	11:
		TON_Abblasdauer(IN := TRUE, PT := Abblasdauer);

		IF 	TON_Abblasdauer.Q
			AND Q_DWORD = 0
		THEN
			state 											:= 10;
		ELSE
			IF 	NOT TOF_Abblastakt.Q 
				AND Q_DWORD <> 0 
			THEN
				TOF_Abblastakt(IN:=TRUE  , PT:= Abblastakt);
				Q_DWORD 									:= 0;
			ELSIF	NOT TOF_Abblastakt.Q 
					AND Q_DWORD = 0 
			THEN
				TOF_Abblastakt(IN:= TRUE , PT:= Abblastakt) ;
				Q_DWORD 									:= SETBIT32(Q_DWORD,i);
			END_IF
			(* Work Timer *)
			TOF_Abblastakt(IN:=FALSE);
		END_IF

	END_CASE
ELSE
	Aktiv 													:= FALSE;
	state 													:= 0;
	Q_DWORD													:= 0;
END_IF

(**********************************************************************************************************)

END_FUNCTION_BLOCK

// ---- POUs/Axis_PTPV3_CoE.TcPOU
FUNCTION_BLOCK Axis_PTPV3_CoE
VAR_OUTPUT CONSTANT
	MIN_JOB													:	INT := 0;
	MAX_JOB													:	INT := 5;
END_VAR
VAR_INPUT
(* Ax Move cmd Parameter *)
	JobId													:	INT := MIN_JOB;
	Job														:	ARRAY[MIN_JOB..MAX_JOB] OF AX_JOB;

(* Axis *)
	ref														:	AXIS_REF; (* siehe Lib TcMc2 *)
	Admin													: 	Ax_AdminCtrl ; (* PTP Ax Control Baustein *)
	para													: 	Ax_Para; (* Achsparameter lesen/schreiben *)
	Motion													:	Ax_MotionCtrl;
	Home													:	Ax_HomingCtrl;
	HMI														:	Ax_HMI;
	Gear				:	Ax_GearCtrl;
	rMasterAxis											:	REFERENCE TO AXIS_REF := 0;
	
(* Ax Optionsmodule *)
	(* Drive *)
	drive													:	Ax_CanOpenDriveEventCtrl;

	(* Error Handling *)
	errorNC													:	Ax_ErrorNCEventCtrl;
                                                    	
	AutoFctCtrl												:	Ax_AutoFctCtrl; (* Softwareendlagen und Refernzierflag ein/ausschalten *)
END_VAR                                             	
VAR_OUTPUT                                          	
	ErrHdl													:	ERROR_HDL;
	EventStatus												:	BYTE;
//	HmiStatus												:	BYTE;
//	startName												:	STRING(10);
//	statusTxt												:	STRING(MAX_STRING_LENGTH);
END_VAR
VAR
	i 														: 	INT;
END_VAR

	(* Axis 																*)
	(************************************************************************)

(* work IO **********************************************************************)


(********************************************************************************)
(* work Admin ctrl 																*)
(********************************************************************************)
	Admin(
		RST			:= , 
		Enable		:= ,
		EnablePos	:= ,
		EnableNeg	:= ,
		BufferMode:= ,
		Override	:= ,
		rAxis		:= Ref,
		ShowNCErrIfDisabled := ,
		EnableOK	=> ,
		Ready		=> ,
		StartRel	=> ,
		Busy		=> ,
		Done		=> ,
		Error		=> ,
		ErrorID		=> );
		
(********************************************************************************)
(* work homing ctrl 															*)
(********************************************************************************)
	Home(
		Execute		:= ,
		Fnc			:= ,
		BufferMode	:= ,
		Mode		:= ,
		AcceptBlockedDrive:= ,
		CalibrationCam:= ,
		Pos			:= ,
		SetPosModeRel:= ,
		SetPosOptions:= ,
		rAxis		:= Ref,
		FNC_HOMING	=> ,
		FNC_HALT	=> ,
		FNC_SETPOS	=> ,
		Active		=> ,
		Done		=> ,
		Busy		=> ,
		CmdAborted	=> ,
		Error		=> ,
		ErrorId		=> ,
		ErrorText	=> );

(********************************************************************************)
(* work moving ctrl 															*)
(********************************************************************************)
	Motion(
		Execute		:= ,
		Fnc			:= ,
		JogFwd		:= ,
		JogBwd		:= ,
		BufferMode	:= ,
		Direction	:= ,
		JogMode		:= ,
		Target		:= ,
		Velo		:= ,
		Jerk		:= ,
		Acc			:= ,
		Dec			:= ,
		MoveOptions:= ,
		rAxis		:= Ref,
		FNC_STOP	=> ,
		FNC_HALT	=> ,
		FNC_MOVE_JOG	=> ,
		FNC_MOVE_ABS	=> ,
		FNC_MOVE_REL	=> ,
		FNC_MOVE_ADD	=> ,
		FNC_MOVE_MOD	=> ,
		FNC_MOVE_VELO	=> ,
		Active		=> ,
		Done		=> ,
		Busy		=> ,
		CmdAborted	=> ,
		Error		=> ,
		ErrorId		=> ,
		ErrorText	=> );

(********************************************************************************)
(* Achse Koppeln 																*)
(********************************************************************************)
(*
	Gear(
		Execute		:= ,
		Fnc			:= ,
		RatioDyn	:= ,
		RatioNumerator:= ,
		RatioDenominator:= ,
		Acc			:= ,
		pMasterAxis1:= ,
		pMasterAxis2:= ,
		pMasterAxis3:= ,
		pMasterAxis4:= ,
		MasterGearRatio1:= ,
		MasterGearRatio2:= ,
		MasterGearRatio3:= ,
		MasterGearRatio4:= ,
		rAxis		:= REF,
		FNC_GEAR_OUT=> ,
		FNC_GEAR_IN=> ,
		FNC_GEAR_IN_DYN=> ,
		FNC_GEAR_IN_MM=> ,
		InGear		=> ,
		Active		=> ,
		Done		=> ,
		Busy		=> ,
		CmdAborted=> ,
		Error		=> ,
		ErrorId		=> ,
		ErrorText	=> );
*)
(********************************************************************************)
(* Parameter																	*)
(*******************************************************************************
	para(
		Execute		:= ,
		Fnc			:= ,
		AxID		:= ref.NcToPlc.AxisId,
		InitDone	=> ,
		Done		=> ,
		Busy		=> ,
		Error		=> );
*)

(******************************************************************************)
(* Hilfsfunktionen der Achse(Setzen,Rücksetzen von Ref.flag und Softwareendl.)*)
(******************************************************************************)
	AutoFctCtrl(
		enable				:= NOT AutoFctCtrl.Error AND Para.InitDone,
		axId				:= ref.NcToPlc.AxisId,
		forceSoftLimit		:= ref.Status.Homed OR para.EncTypAbs = 1, (* nicht referenziert oder Encodertyp Abs. *)
		forceCalibration	:= , //Siehe Abblikation 
		Status				=> ,
		Busy				=> ,
		Error				=> ,
		ErrorId				=> );

(********************************************************************************)
(* Error NC																		*)
(********************************************************************************)
	IF Admin.Error
	THEN
		ErrHdl.id 		:= UDINT_TO_DINT(Admin.ErrorId);
		ErrHdl.fnc		:= 'Admin';
		ErrHdl.text		:= Admin.ErrorText;
		ErrHdl.flag		:= TRUE;
	ELSIF Motion.Error
	THEN
		ErrHdl.id 		:= UDINT_TO_DINT(Motion.ErrorId);
		ErrHdl.fnc		:= 'Motion';
		ErrHdl.text		:= Motion.ErrorText;
		ErrHdl.flag		:= TRUE;
	ELSIF Home.Error
	THEN
		ErrHdl.id 		:= UDINT_TO_DINT(Home.ErrorId);
		ErrHdl.fnc		:= 'Home';
		ErrHdl.text		:= Home.ErrorText;
		ErrHdl.flag		:= TRUE;

(*	ELSIF Gear.Error
	THEN
		ErrHdl.id 		:= UDINT_TO_DINT(gear.ErrorId);
		ErrHdl.fnc		:= 'Gear';
		ErrHdl.text		:= Gear.ErrorText;
		ErrHdl.flag		:= TRUE;
*)
	ELSE
		ErrHdl.Reset();
	END_IF
	
	errorNC(
		Enable			:=	Admin.EnableOK,
		InAck			:= NOT Errhdl.flag AND errorNC.StatusByte <> 0 OR Admin.RST,
		Name			:= para.Name,
		SourceId		:= (* Default *) ,
		rAxis			:= ref,
		AxErrorId		:= DINT_TO_UDINT(ErrHdl.Id),
		CmdAborted		:= ,
		StatusByte		=> ,
		SOURCE_AXIS		=> );
		
(********************************************************************************)
(* Drive 																		*)
(********************************************************************************)
	drive(
		EnableEvent		:= , 
		InAck			:= errorNC.InAck, 
		Name			:= para.Name, 
		ErrorEndlagePos:= , 
		ErrorEndlageNeg:= , 
		ErrorSchutzschalter:= , 
		rAxis			:= ref, 
		Busy			=> , 
		Error			=> , 
		ErrorId			=> , 
		Fault			=> , 
		Ready			=> , 
		LiveCountTimeout=> , 
		LiveCount		=> , 
		RT_StatusChanged=> , 
		CanNodeSTATE	=> , 
		EventStatusByte	=> , 
		SOURCE_DRIVES_CAN=> );
		
(* Event Status *****************************************************************)
	EventStatus																:= 	errorNC.StatusByte
																				OR Drive.EventStatusByte;
		
(* Check start arr pos **********************************************************)
	CheckTargetPos();

(********************************************************************************)
(* Hmi Axis				 														*)
(********************************************************************************)
	HMI(Motion := Motion);
	
	Gear(
	FNC_GEAR_OUT=> , 
	FNC_GEAR_IN=> , 
	FNC_GEAR_IN_DYN=> , 
	FNC_GEAR_IN_MM=> , 
	Execute:= , 
	Fnc:= , 
	RatioDyn:= , 
	RatioNumerator:= , 
	RatioDenominator:= , 
	Acc:= , 
	Options:= , 
	rMasterAxis1:=rMasterAxis , 		//直接写
	rMasterAxis2:= , 
	rMasterAxis3:= , 
	rMasterAxis4:= , 
	MasterGearRatio1:= , 
	MasterGearRatio2:= , 
	MasterGearRatio3:= , 
	MasterGearRatio4:= , 
	rAxis:= ref, 
	Active=> , 
	Done=> , 
	Busy=> , 
	CmdAborted=> , 
	Error=> , 
	ErrorId=> , 
	ErrorText=> );
	
	
(*
	HmiStatus.0 := ref.Status.NegativeDirection;
	HmiStatus.1 := ref.Status.PositiveDirection;
	HmiStatus.2 := ref.Status.InTargetPosition  ;
	HmiStatus.3 := ref.Status.Homed;
	HmiStatus.4 := Admin.EnableNeg; 
	HmiStatus.5 := Admin.EnablePos;
	HmiStatus.6 := Admin.Ready;
	HmiStatus.7 := ErrHdl.flag;
*)
(* Set Status Txt ***************************************************************)
(*	IF Pulse._1s.RT THEN
		statusTxt := CONCAT(para.Name,' Id:');
		statusTxt := CONCAT(statusTxt,DWORD_TO_STRING(ref.NcToPlc.AxisId));
		statusTxt := CONCAT(statusTxt,SEL(ctrl.Ready,',NOT Ready,Istpos:',',Ready,Istpos:'));
		statusTxt := CONCAT(statusTxt,LREAL_TO_FMTSTR(ctrl.ActPos, 2, TRUE));
		statusTxt := CONCAT(statusTxt,',Target:');
		statusTxt := CONCAT(statusTxt,LREAL_TO_FMTSTR(ctrl.Target, 2, TRUE));
		(* Zeilenwechsel *)
		statusTxt := CONCAT(statusTxt,'$r');
		(* ------------- *)
		statusTxt := CONCAT(statusTxt,SEL(ctrl.NotMoving,SEL(ref.Status.PositiveDirection,',Moving NEG,StartId:',',Moving POS,StartId:'),',NOT Moving,StartId:'));
		statusTxt := CONCAT(statusTxt,INT_TO_STRING(StartID));
		statusTxt := CONCAT(statusTxt,',ErrorId:');
		statusTxt := CONCAT(statusTxt,DINT_TO_STRING(ctrl.ErrHdl.id));
		statusTxt := CONCAT(statusTxt,',Cmd:');
		statusTxt := CONCAT(statusTxt,INT_TO_STRING(ctrl.Cmd));
		statusTxt := CONCAT(statusTxt,',ActCmd:');
		statusTxt := CONCAT(statusTxt,INT_TO_STRING(ctrl.Actcmd));
	END_IF
*)


(***********************************************************************************************)

METHOD PUBLIC CheckTargetPos
VAR_INPUT
END_VAR
FOR i := MIN_JOB TO MAX_JOB DO
	IF Job[i].Fnc = 6 THEN
		Job[i].InTarget := REF.Status.NotMoving
									AND(
									REF.NcToPlc.ModuloActPos >= Job[i].Target - para.Zielfenster
									AND REF.NcToPlc.ModuloActPos <= Job[i].Target + para.Zielfenster
									OR
									(MODABS(Job[i].Target,para.ModuloFaktor) <= 0 + para.Zielfenster
									OR MODABS(Job[i].Target,para.ModuloFaktor) >= para.ModuloFaktor - para.Zielfenster)
									AND(
									REF.NcToPlc.ModuloActPos >= para.ModuloFaktor - para.Zielfenster
									OR REF.NcToPlc.ModuloActPos <= 0 + para.Zielfenster));

		Job[i].InPosWindow	:= REF.NcToPlc.ModuloActPos >= Job[i].Target - para.Posfenster
									AND REF.NcToPlc.ModuloActPos <= Job[i].Target + para.Posfenster
									OR
									(MODABS(Job[i].Target,para.ModuloFaktor) <= 0 + para.Posfenster
									OR MODABS(Job[i].Target,para.ModuloFaktor) >= para.ModuloFaktor - para.Posfenster)
									AND(
									REF.NcToPlc.ModuloActPos >= para.ModuloFaktor - para.Posfenster
									OR REF.NcToPlc.ModuloActPos <= 0 + para.Posfenster);
	ELSE
		Job[i].InTarget := REF.Status.NotMoving
									AND REF.NcToPlc.ActPos >= Job[i].Target - para.Zielfenster
									AND REF.NcToPlc.ActPos <= Job[i].Target + para.Zielfenster ;

		Job[i].InPosWindow	:= REF.NcToPlc.ActPos >= Job[i].Target - para.Posfenster
									AND REF.NcToPlc.ActPos <= Job[i].Target + para.Posfenster;
	END_IF
END_FOR
END_METHOD

METHOD PUBLIC NoAction : BOOL //Result = Busy of home , gear , motion , ....
VAR_INPUT
END_VAR
home.Execute	:= FALSE;
//gear.Execute	:= FALSE;
Motion.Execute	:= FALSE;
Motion.JogBwd	:= FALSE;
Motion.JogFwd	:= FALSE;
Gear.Execute	:=FALSE;

NoAction 		:= NOT home.Busy
					AND NOT gear.Busy
					and not Motion.Busy;
END_METHOD

METHOD PUBLIC reset
VAR_INPUT
END_VAR
Admin.Reset(FALSE);
drive.Ack();
errorNC.Ack();
END_METHOD

METHOD PUBLIC StartMotion
VAR_INPUT
	JobID			:	int ;
END_VAR
THIS^.JobID		:= Jobid;

IF JobID >= MIN_JOB AND JobId <= MAX_JOB
THEN
	CheckTargetPos();
//	startName				:= Job[Jobid].name;
	Motion.Fnc 				:= Job[Jobid].Fnc;
	Motion.BufferMode 		:= Job[Jobid].BufferMode;
	Motion.Direction 		:= Job[Jobid].Direction;
	Motion.Target 			:= Job[Jobid].Target;
	Motion.Velo 			:= Job[Jobid].Velo;
	Admin.Override 			:= Job[Jobid].Override;
	Motion.Acc		 		:= Job[Jobid].Acc;
	Motion.Dec				:= Job[Jobid].Dec;
	Motion.Jerk	 			:= Job[Jobid].Jerk;
	MOtion.Execute			:= TRUE;
END_IF
END_METHOD

END_FUNCTION_BLOCK

// ---- POUs/PTP/01_Base/Ax_MotionCtrl.TcPOU
{attribute 'no_check'}
FUNCTION_BLOCK Ax_MotionCtrl (* Achse reseten,BTB schalten, starten und stoppen *)
(* A C H T U N G !!!
	For performance reasons the MC-function-blocks MC_MoveRelative, MC_MoveAdditive, MC_MoveVelocity and 
	MC_MoveModulo are commented out insed the declaration.
	If needed, the comment-signs can be removed.

	Alle Bausteine sind schon ausprogrammiert und können in vollem Umfang benutzt werden.
	(MC_MoveAbsolute ->  MC_MoveRelative mit BufferMode-Aborting -> MC_MoveAdditive mit BufferMode-MC_BlendingLow ... 

*)  
VAR_OUTPUT CONSTANT
	FNC_HALT												:	INT := 0;
	FNC_STOP												:	INT := 1;
	FNC_MOVE_JOG											:	INT := 2;
	FNC_MOVE_ABS											:	INT := 3;
	FNC_MOVE_REL											:	INT := 4;
	FNC_MOVE_ADD											:	INT := 5;
	FNC_MOVE_MOD											:	INT := 6;
	FNC_MOVE_VELO											:	INT := 7;
END_VAR
VAR_INPUT
	Execute													:	BOOL := FALSE;
	Fnc														:	INT (FNC_HALT..FNC_MOVE_VELO) := FNC_HALT;
	JogFwd													:	BOOL := FALSE;
	JogBwd													:	BOOL	:= FALSE;
	BufferMode												:	MC_BufferMode := MC_Aborting;(* 	MC_Aborting,
																											MC_Buffered,
																											MC_BlendingLow,
																											MC_BlendingPrevious,
																											MC_BlendingNext,
																											MC_BlendingHigh *)
	Direction												:	MC_Direction := MC_POSITIVE_DIRECTION;	(*	MC_POSITIVE_DIRECTION,
																														   MC_SHORTeSTATE.WAY,
																														   MC_NEGATIVE_DIRECTION,
																														   MC_CURRENT_DIRECTION *)
	JogMode													:	E_JogMode := MC_JOGMODE_STANDARD_SLOW;	(*	MC_JOGMODE_STANDARD_SLOW
																															MC_JOGMODE_STANDARD_FAST
																															MC_JOGMODE_CONTINOUS
																															MC_JOGMODE_INCHING 
																															MC_JOGeMODE.INCHING_MODULO *)
	Target													:	LREAL; (* Zielposition *)
	Velo														: 	LREAL; (* Zielgeschwindigkeit *)
	Jerk														:	LREAL := 0.0; (* Bei 0 werden wird der Ruck aus dem TCManager uebernommen *)
	Acc														:	LREAL := 0.0; (* Bei 0 werden wird die Beschleunigung aus dem TCManager uebernommen *)
	Dec														:	LREAL := 0.0; (* Bei 0 werden wird die Verzoegerung aus dem TCManager uebernommen *)
	MoveOptions												:	ST_MoveOptions;
	rAxis														:	REFERENCE TO AXIS_REF := 0;
END_VAR                     								
VAR_IN_OUT                  								
END_VAR                     								
VAR_OUTPUT                  								
	Active													:	BOOL;
	Done													:	BOOL;
	Busy													:	BOOL;
	CmdAborted												:	BOOL;
	Error													:	BOOL;
	ErrorId													:	UDINT;
	ErrorText												:	STRING(40);
END_VAR
VAR
(* Zwischenspeicher **************************************************************************)
	MemFnc													:	INT := -1;
	MemFncAct												:	INT := -1;
	MCFctTxt												:	STRING(25);
	TrigID													:	INT := 2; (* um mit Trig 1 zu starten *)
	MemBufferMode											:	MC_BufferMode;
	ActSetTarget											:	LREAL;
	ActSetVelo												:	LREAL;
	BusyIntern												:	BOOL;

(* Timer *)

(* Trigger *)
	rtExecute												:	R_TRIG;
	rtExecuteMethod											:	R_TRIG;

(* Instanzierung der MC Bausteine *******************************************************)
	MC_Halt													: 	MC_Halt;
	MC_Stop													: 	MC_Stop;
	MC_MoveVeloPreTrig										: 	MC_MoveVelocity;
	MC_Jog													: 	MC_Jog;

(* Durch entfernen der Kommentarsymbole koennen noch weitere benötigte MC_Move Varianten
	mit ins Programm genommen werden 
*)
	MC_MoveAbsolute											: 	ARRAY[1..2] OF MC_MoveAbsolute;
	MC_MoveModulo											: 	ARRAY[1..2] OF MC_MoveModulo;
	MC_MoveRelative											: 	ARRAY[1..2] OF MC_MoveRelative;
	MC_MoveAdditive											: 	ARRAY[1..2] OF MC_MoveAdditive; 
	MC_MoveVelocity											: 	ARRAY[1..2] OF MC_MoveVelocity; 

(* Dummy Speicher **********************************************************)
	i														: INT := 0 ;

(* Skalierungsfaktor ermitteln *********************************************
	Skalierungsfaktor von 0.1 eintragen. Istpositon "Anfang" merken.
	Antrieb um einen realen Wert "X" mm verfahren. Differenz der
	momentanen Istposition zur Istposition "Anfang" ermitteln.
	SKalierungsfaktor =		realer Fahrweg 
							---------------------------
							Differenz der Istpositionen
*)
END_VAR

	(****************************************************************************************)
	(*																						*)
	(*		B E C K H O F F   N E W   A U T O M A T I O N   T E C H N O L O G Y    			*)
	(*																						*)
	(*		Eiserstr.5	D-33415 Verl	Germany	phone:	+49-5246-0	www.Beckhoff.Com		*)
    (*																						*)
    (*		Bausteinbeschreibung	:	Ax Move Ctrl										*)
	(*		TwinCAT-Version			:	3.x or higher										*)
	(*		Lib						:	TcMC2.lib Newest Version!							*)
	(*		Version					:	V1.2												*)
 	(*		Autor					:	Daniel Schlingmann									*)
	(*																						*)
	(*		Changelog:																		*)
	(*		12.07.14	-	Kein Signal CmdAborted von MC_Jog wenn Software Endl erreicht	*)
	(****************************************************************************************)

(* Execute ***************************************************************************************)
	rtExecute(CLK := Execute XOR(JogBwd AND NOT JogFwd OR JogFwd AND NOT JogBwd));
	
	IF rtExecute.Q
	THEN
		MemFnc 												:= SEL(JogBwd OR JogFwd, Fnc, FNC_MOVE_JOG) ;
		Busy												:= TRUE;
		Done												:= FALSE;
		Active												:= FALSE;
		Error												:= FALSE;
		ErrorID												:= 0;
		CmdAborted											:= FALSE;
		ErrorText											:= '';
	END_IF

(* Call Method ***********************************************************************************)
	CASE MemFnc OF
	FNC_STOP												:	Stop(Execute);
	FNC_HALT												:	Halt(Execute);
	FNC_MOVE_JOG											:	MoveJog(Execute);
	FNC_MOVE_ABS											:	MoveAbs(Execute);
	FNC_MOVE_REL											:	MoveRel(Execute);
	FNC_MOVE_ADD											:	MoveAdd(Execute);
	FNC_MOVE_MOD											:	MoveMod(Execute);
	FNC_MOVE_VELO											:	MoveVelo(Execute);
	-1:
		IF NOT Execute
		THEN
			Busy											:= FALSE;
			Done											:= FALSE;
			Error											:= FALSE;
			ErrorID											:= 0;
			Active											:= FALSE;
			CmdAborted										:= FALSE;
			ErrorText										:= '';
		END_IF
	ELSE
		Busy												:= FALSE;
		Done												:= FALSE;
		Active												:= FALSE;
		Error												:= Execute;
		ErrorID												:= 1803;
		CmdAborted											:= FALSE;
		ErrorText											:= CONCAT('invalid parameter value(s) Fnc no: ' , INT_TO_STRING(MemFnc));
	END_CASE

(*************************************************************************************************)

METHOD PRIVATE _MCIntern
VAR_INPUT
END_VAR
(* Internal MC Action											*)
(****************************************************************)

(* Check Pointer **********************************************************************)
IF NOT __ISVALIDREF(rAxis) 
THEN
	Busy													:= NOT Error;
	Error													:= TRUE;
	ErrorId													:= 16#4B30;
	CmdAborted												:= FALSE;
	Done														:= FALSE;
	Active													:= FALSE;
	ErrorText												:= 'Reference rAxis invalid (0)';
	MemFnc													:= SEL(Execute , -1 ,MemFnc); 
	RETURN;
END_IF

(* flag Execute ***********************************************************************)
	rtExecuteMethod(CLK := Execute OR rtExecute.Q);
	IF rtExecuteMethod.Q
	THEN
		MC_Stop.Execute										:= FALSE;
		MC_Halt.Execute										:=	FALSE;
		MC_MoveVeloPreTrig.Execute							:= FALSE;
		MC_MoveModulo[1].Execute 							:= MC_MoveModulo[2].Execute	:= FALSE;
		MC_MoveAbsolute[1].Execute							:= MC_MoveAbsolute[2].Execute	:= FALSE;
		MC_MoveRelative[1].Execute 							:= MC_MoveRelative[2].Execute := FALSE; 
		MC_MoveAdditive[1].Execute 							:= MC_MoveAdditive[2].Execute := FALSE; 
		MC_MoveVelocity[1].Execute 							:= MC_MoveVelocity[2].Execute := FALSE; 
		BusyIntern											:= FALSE;
		MemFncAct 											:= MemFnc;
	END_IF

(* ctrl programm ******************************************************************************)
	CASE MemFncAct OF
	-1: ; //No Fnc started
	FNC_STOP:
		MC_Stop.Execute										:=	Execute; (* Achse Locked solange Stop noch ansteht *)
		MC_Stop.Deceleration 								:= Dec;
		MC_Stop.Jerk 										:= Jerk;
		MC_Stop.Options 									:= MoveOptions;

	FNC_HALT:
		MC_Halt.Execute										:=	NOT MC_Stop.Busy AND Execute; (* Execute if axis is not locked *)
		MC_Halt.BufferMode									:= BufferMode;
		MC_Halt.Deceleration 								:= Dec;
		MC_Halt.Jerk 										:= Jerk;
		MC_Halt.Options 									:= MoveOptions;
		BusyIntern											:= MC_Stop.Busy;

	FNC_MOVE_JOG:
		IF(Execute OR JogBwd OR JogFwd OR MC_Halt.Busy) (* new cmd or stop last cmd busy *)
			AND NOT rAxis.NcToPlc.StateDWord.2  (* NotMoving *)
			AND NOT MC_Jog.Busy (* not if Mc_Jog running *)
			AND NOT rAxis.NcToPlc.StateDWord.5 (* Protected *) (* not if axis coupled or in NCI group *)
			AND NOT MC_Halt.Error AND NOT MC_Halt.CommandAborted
		THEN
			MC_Halt.Execute									:=	TRUE;
			MC_Halt.BufferMode								:= MC_Aborting;
			MC_Halt.Deceleration 							:= Dec;
			MC_Halt.Jerk 									:= Jerk;
			MC_Halt.Options 								:= MoveOptions;
			BusyIntern										:= TRUE;
		ELSE
			MC_Jog.JogBackwards								:= NOT MC_Stop.Busy AND (JogBwd XOR Execute AND Direction = MC_NEGATIVE_DIRECTION);
			MC_Jog.JogForward								:= NOT MC_Stop.Busy AND (JogFwd XOR Execute AND Direction = MC_POSITIVE_DIRECTION);
			MC_Jog.Mode										:= JogMode;
			MC_Jog.Position 								:= Target;
			MC_Jog.Velocity 								:= Velo;
			MC_Jog.Acceleration 							:= Acc;
			MC_Jog.Deceleration 							:= Dec;
			MC_Jog.Jerk 									:= Jerk;
			MC_Halt.Execute									:=	FALSE;
			BusyIntern										:= MC_Stop.Busy;
		END_IF

	FNC_MOVE_ABS..FNC_MOVE_VELO:
		IF MC_Stop.Busy
			OR rAxis.NcToPlc.StateDWord.29 (* MotionCommandsLocked *)
			OR MC_Jog.Busy
		THEN (* Solange hier rein bis Achse wieder frei und Stop nicht mehr Busy *)
			BusyIntern										:= TRUE;

		ELSIF rAxis.NcToPlc.StateDWord.24 (* CmdBuffered *) 
		THEN (* this section is for aborting a buffered running axis *)
			IF NOT MC_MoveVeloPreTrig.Execute
				AND BufferMode = MC_Aborting
				AND(
				rtExecuteMethod.Q (* new cmd with MC_Aborting zu break up current and buffered cmd *)
				OR 		(* or break up current and buffered cmd with new targetpos. *)
				Execute
				AND (Busy OR Done OR CmdAborted) (* dont restart if error is active *)
				AND (ActSetTarget <> Target))
			THEN
				TrigID 										:= 0;
				MC_MoveVeloPreTrig.Execute 					:= TRUE;
				MC_MoveVeloPreTrig.BufferMode 				:= MC_Aborting;
				MC_MoveVeloPreTrig.Velocity 				:= Velo;
				IF rAxis.NcToPlc.StateDWord.10 (* NegativeDirection *) 
				THEN
					MC_MoveVeloPreTrig.Direction 			:= MC_NEGATIVE_DIRECTION;
				ELSE
					MC_MoveVeloPreTrig.Direction 			:= MC_POSITIVE_DIRECTION;
				END_IF
				BusyIntern									:= TRUE;
			ELSE
				;
			END_IF

		ELSE (* ready for start/restart (MC_MoveVeloPreTrig is active) *)
			IF rtExecuteMethod.Q (* new cmd *)
				OR TrigID = 0 (* new cmd with Buffermode aborted *)
				OR(	Execute
				AND (Busy OR Done OR CmdAborted) (* dont restart if error is active *)
				AND (ActSetTarget <> Target OR ActSetVelo <> Velo AND BufferMode = MC_Aborting)) (* restart only with new velo if bufferMode = Aborting *)
			THEN (* new cmd *)
				(* Cancel MoveVeloPreTrig block *)
				IF TrigID = 0 THEN
					MemBufferMode 							:= MC_Aborting;
				ELSE
					MemBufferMode						 	:= BufferMode;
				END_IF

				(* change TrigID *)
				IF TrigID <> 1 THEN
					TrigID 									:= 1;
				ELSE
					TrigID 									:= 2;
				END_IF

				(* Save Act. target and velo *)
				ActSetTarget 								:= Target;
				ActSetVelo 									:= Velo;

				(* Init MC-Blocks *)
				MC_MoveModulo[1].Execute 					:= MC_MoveModulo[2].Execute	:= FALSE;
				MC_MoveAbsolute[1].Execute					:= MC_MoveAbsolute[2].Execute	:= FALSE;
				MC_MoveRelative[1].Execute 					:= MC_MoveRelative[2].Execute := FALSE; 
				MC_MoveAdditive[1].Execute 					:= MC_MoveAdditive[2].Execute := FALSE; 
				MC_MoveVelocity[1].Execute 					:= MC_MoveVelocity[2].Execute := FALSE; 
			END_IF

			CASE MemFncAct OF
			FNC_MOVE_ABS:(* Absolute *);
				MC_MoveAbsolute[TrigID].Execute				:= Execute OR BusyIntern;
				MC_MoveAbsolute[TrigID].BufferMode 			:= MemBufferMode;
				MC_MoveAbsolute[TrigID].Position 			:= Target;
				MC_MoveAbsolute[TrigID].Velocity 			:= Velo;
				MC_MoveAbsolute[TrigID].Acceleration 		:= Acc;
				MC_MoveAbsolute[TrigID].Deceleration 		:= Dec;
				MC_MoveAbsolute[TrigID].Jerk 				:= Jerk;
				MC_MoveAbsolute[TrigID].Options 			:= MoveOptions;

			FNC_MOVE_MOD:(* Modulo *);
				MC_MoveModulo[TrigID].Execute				:= Execute OR BusyIntern;
				MC_MoveModulo[TrigID].BufferMode 			:= MemBufferMode;
				MC_MoveModulo[TrigID].Position 				:= Target;
				MC_MoveModulo[TrigID].Direction 			:= Direction;
				MC_MoveModulo[TrigID].Velocity 				:= Velo;
				MC_MoveModulo[TrigID].Acceleration 			:= Acc;
				MC_MoveModulo[TrigID].Deceleration 			:= Dec;
				MC_MoveModulo[TrigID].Jerk 					:= Jerk;
				MC_MoveModulo[TrigID].Options 				:= MoveOptions;
			
			FNC_MOVE_REL: (* Relativ *)
				MC_MoveRelative[TrigID].Execute				:= Execute OR BusyIntern;
				MC_MoveRelative[TrigID].BufferMode 			:= MemBufferMode;
				MC_MoveRelative[TrigID].Distance 			:= Target;
				MC_MoveRelative[TrigID].Velocity 			:= Velo;
				MC_MoveRelative[TrigID].Acceleration 		:= Acc;
				MC_MoveRelative[TrigID].Deceleration	 	:= Dec;
				MC_MoveRelative[TrigID].Jerk 				:= Jerk;
				MC_MoveRelative[TrigID].Options 			:= MoveOptions;
		
			FNC_MOVE_ADD:(* Rel.Additive *);
				MC_MoveAdditive[TrigID].Execute				:= Execute OR BusyIntern;
				MC_MoveAdditive[TrigID].BufferMode 			:= MemBufferMode;
				MC_MoveAdditive[TrigID].Distance 			:= Target;
				MC_MoveAdditive[TrigID].Velocity 			:= Velo;
				MC_MoveAdditive[TrigID].Acceleration	 	:= Acc;
				MC_MoveAdditive[TrigID].Deceleration	 	:= Dec;
				MC_MoveAdditive[TrigID].Jerk 				:= Jerk;
				MC_MoveAdditive[TrigID].Options 			:= MoveOptions;
			
			FNC_MOVE_VELO:(* Velocity *);
				MC_MoveVelocity[TrigID].Execute				:= Execute OR BusyIntern;
				MC_MoveVelocity[TrigID].BufferMode 			:= MemBufferMode;
				MC_MoveVelocity[TrigID].Direction 			:= Direction;
				MC_MoveVelocity[TrigID].Velocity 			:= Velo;
				MC_MoveVelocity[TrigID].Acceleration 		:= Acc;
				MC_MoveVelocity[TrigID].Deceleration 		:= Dec;
				MC_MoveVelocity[TrigID].Jerk 				:= Jerk;
				MC_MoveVelocity[TrigID].Options 			:= MoveOptions;
			
			ELSE
				MC_Halt.Execute								:=	TRUE; // axis locked as long as Stop is set 
				Error										:= TRUE;
				ErrorId										:= 16#1803;
				ErrorText									:= CONCAT('invalid parameter value(s) - Fnc no ', INT_TO_STRING(MemFncAct)) ;
			END_CASE

			(* Reset busy intern *)
			MC_MoveVeloPreTrig.Execute 						:= FALSE;
			BusyIntern										:= FALSE;
		END_IF
	ELSE
		MC_Halt.Execute										:=	TRUE; // axis locked as long as Stop is set
		Error												:= TRUE;
		ErrorId												:= 16#1803;
		ErrorText											:= CONCAT('invalid parameter value(s) - Fnc no ', INT_TO_STRING(MemFncAct)) ;
	END_CASE

(****************************************************************************)
(* Work MC Blocks 															*)
(****************************************************************************)

	(* Halt/Stop *)
	MC_Stop(Axis	:= rAxis);
	MC_Halt(Axis	:= rAxis);

	(* Jog *)
	IF MC_Jog.JogBackwards OR MC_Jog.JogForward OR MC_Jog.Busy
		OR MC_Jog.Done OR MC_Jog.Active
		OR MC_Jog.CommandAborted OR MC_Jog.Error
	THEN
		MC_Jog( Axis :=	rAxis);
		MC_Jog.JogBackwards									:= FALSE;
		MC_Jog.JogForward									:= FALSE;
	END_IF

	(* Positionierungen ********************************************)
	(* MC Move Velo PreTrig 1 *)
	IF MC_MoveVeloPreTrig.Execute OR MC_MoveVeloPreTrig.Busy
		OR MC_MoveVeloPreTrig.InVelocity OR MC_MoveVeloPreTrig.Active
		OR MC_MoveVeloPreTrig.CommandAborted OR MC_MoveVeloPreTrig.Error
	THEN
		MC_MoveVeloPreTrig(Axis	:=	rAxis);
	END_IF

	(* Run MC *)
	IF MC_MoveAbsolute[1].Execute OR MC_MoveAbsolute[1].Busy
		OR MC_MoveAbsolute[1].Done OR MC_MoveAbsolute[1].Active
		OR MC_MoveAbsolute[1].CommandAborted OR MC_MoveAbsolute[1].Error
	THEN
		MC_MoveAbsolute[1]( Axis	:=	rAxis);
	END_IF

	IF MC_MoveModulo[1].Execute OR MC_MoveModulo[1].Busy
		OR MC_MoveModulo[1].Done OR MC_MoveModulo[1].Active
		OR MC_MoveModulo[1].CommandAborted OR MC_MoveModulo[1].Error
	THEN
		MC_MoveModulo[1](Axis	:=	rAxis);
	END_IF
	
	IF MC_MoveRelative[1].Execute OR MC_MoveRelative[1].Busy
		OR MC_MoveRelative[1].Done OR MC_MoveRelative[1].Active
		OR MC_MoveRelative[1].CommandAborted OR MC_MoveRelative[1].Error
	THEN
		MC_MoveRelative[1](Axis	:=	rAxis);
	END_IF
	
	IF MC_MoveAdditive[1].Execute OR MC_MoveAdditive[1].Busy
		OR MC_MoveAdditive[1].Done OR MC_MoveAdditive[1].Active
		OR MC_MoveAdditive[1].CommandAborted OR MC_MoveAdditive[1].Error
	THEN
		MC_MoveAdditive[1](Axis	:=	rAxis);
	END_IF
	
	IF MC_MoveVelocity[1].Execute OR MC_MoveVelocity[1].Busy
		OR MC_MoveVelocity[1].Active OR MC_MoveVelocity[1].InVelocity
		OR MC_MoveVelocity[1].CommandAborted OR MC_MoveVelocity[1].Error
	THEN
		MC_MoveVelocity[1](Axis	:=	rAxis);
	END_IF

	(* MC Move Velo PreTrig 2 **************************************)
	(* Run Trig 2 *)
	IF MC_MoveAbsolute[2].Execute OR MC_MoveAbsolute[2].Busy
		OR MC_MoveAbsolute[2].Done OR MC_MoveAbsolute[2].Active
		OR MC_MoveAbsolute[2].CommandAborted OR MC_MoveAbsolute[2].Error
	THEN
		MC_MoveAbsolute[2](Axis	:=	rAxis);
	END_IF

	IF MC_MoveModulo[2].Execute OR MC_MoveModulo[2].Busy
		OR MC_MoveModulo[2].Done OR MC_MoveModulo[2].Active
		OR MC_MoveModulo[2].CommandAborted OR MC_MoveModulo[2].Error
	THEN
		MC_MoveModulo[2](Axis	:=	rAxis);
	END_IF

	
	IF MC_MoveRelative[2].Execute OR MC_MoveRelative[2].Busy
		OR MC_MoveRelative[2].Done OR MC_MoveRelative[2].Active
		OR MC_MoveRelative[2].CommandAborted OR MC_MoveRelative[2].Error
	THEN
		MC_MoveRelative[2](Axis	:=	rAxis);
	END_IF
	
	IF MC_MoveAdditive[2].Execute OR MC_MoveAdditive[2].Busy
		OR MC_MoveAdditive[2].Done OR MC_MoveAdditive[2].Active
		OR MC_MoveAdditive[2].CommandAborted OR MC_MoveAdditive[2].Error
	THEN
		MC_MoveAdditive[2](Axis	:=	rAxis);
	END_IF

	
	IF MC_MoveVelocity[2].Execute OR MC_MoveVelocity[2].Busy
		OR MC_MoveVelocity[2].Active OR MC_MoveVelocity[2].InVelocity
		OR MC_MoveVelocity[2].CommandAborted OR MC_MoveVelocity[2].Error
	THEN
		MC_MoveVelocity[2](Axis	:=	rAxis);
	END_IF

(******************************************************************************)
(* Ctrl Status 																					*)
(******************************************************************************)
	IF MemFncAct = FNC_STOP
	THEN (* as long as MC_Stop running the axis is locked *)
		MCFctTxt											:= 'MC_STOP';
		Done 												:= MC_Stop.Done;
		Busy 												:= MC_Stop.Busy;
		Active 												:= MC_Stop.Active;
		CmdAborted 											:= MC_Stop.CommandAborted;
		Error												:=	MC_Stop.Error;
		ErrorId												:= MC_Stop.ErrorId;
		ErrorText											:= SEL(Error , '' ,  CONCAT('Error MC_STOP id: ',  UDINT_TO_STRING(Errorid)));

	ELSIF MemFncAct = FNC_HALT
	THEN
		MCFctTxt											:= 'MC_HALT';
		Done 												:= MC_Halt.Done;
		Busy 												:= MC_Halt.Busy;
		Active 												:= MC_Halt.Active;
		CmdAborted 	 										:= MC_Halt.CommandAborted;
		Error												:=	MC_Halt.Error;
		ErrorId												:= MC_Halt.ErrorId;
		ErrorText											:= SEL(Error , '' ,  CONCAT('Error MC_HALT id: ',  UDINT_TO_STRING(Errorid)));

	ELSIF BusyIntern
	THEN
		MCFctTxt											:= CONCAT('BUSY INTERN at Fnc no: ', INT_TO_STRING(MemFncAct));
		Busy												:= BusyIntern;
		Done 												:= FALSE;
		Active 												:= FALSE;
		CmdAborted 											:= FALSE;
		Error												:=	FALSE;
		ErrorId												:= 0;
		ErrorText											:= '';

	ELSIF MemFncAct = FNC_MOVE_JOG
	THEN
		MCFctTxt											:= 'MC_JOG';
		Done 												:= MC_Jog.Done;
		Busy 												:= MC_Jog.Busy;
		Active 												:= MC_Jog.Active;
		CmdAborted 	 										:= MC_Jog.CommandAborted AND NOT rAxis.NcToPlc.StateDWord.26 AND NOT rAxis.NcToPlc.StateDWord.27  (* Software limit exceeded *) ;
		Error												:=	MC_Jog.Error;
		ErrorId												:= MC_Jog.ErrorId;
		ErrorText											:= SEL(Error , '' ,  CONCAT('Error MC_JOG id: ',  UDINT_TO_STRING(Errorid)));

	ELSIF MC_MoveVeloPreTrig.Execute
		OR TrigID = 0
	THEN (* Pretrig Block *)
		MCFctTxt											:= 'MC_MoveVeloPreTrig';
		Done												:= FALSE;
		Busy												:= MC_MoveVeloPreTrig.Busy;
		Active 												:= MC_MoveVeloPreTrig.Active;
		CmdAborted 	 										:= MC_MoveVeloPreTrig.CommandAborted;
		Error												:=	MC_MoveVeloPreTrig.Error;
		ErrorId												:= MC_MoveVeloPreTrig.ErrorId;
		ErrorText											:= SEL(Error , '' ,  CONCAT('Error MC_MoveVeloPreTrig id: ',  UDINT_TO_STRING(Errorid)));

	ELSIF MemFncAct = FNC_MOVE_ABS
	THEN (* Absolut *)
		MCFctTxt											:= CONCAT('MC_MoveAbs TrigID No:',INT_TO_STRING(TrigID));
		Done 												:= MC_MoveAbsolute[TrigID].Done;
		Busy 												:= MC_MoveAbsolute[TrigID].Busy;
		Active 												:= MC_MoveAbsolute[TrigID].Active;
		CmdAborted 	 										:= MC_MoveAbsolute[TrigID].CommandAborted;
		Error												:=	MC_MoveAbsolute[TrigID].Error;
		ErrorId												:= MC_MoveAbsolute[TrigID].ErrorId;
		ErrorText											:= SEL(Error , '' ,  CONCAT('Error MC_MoveAbsolute id: ',  UDINT_TO_STRING(Errorid)));
	
	ELSIF MemFncAct = FNC_MOVE_MOD
	THEN (* Modulo *)
		MCFctTxt											:= CONCAT('MC_MoveModulo TrigID No:',INT_TO_STRING(TrigID));
		Done 												:= MC_MoveModulo[TrigID].Done;
		Busy 												:= MC_MoveModulo[TrigID].Busy;
		Active 												:= MC_MoveModulo[TrigID].Active;
		CmdAborted 											:= MC_MoveModulo[TrigID].CommandAborted;
		Error												:=	MC_MoveModulo[TrigID].Error;
		ErrorId												:= MC_MoveModulo[TrigID].ErrorId;
		ErrorText											:= SEL(Error , '' ,  CONCAT('Error MC_MoveModulo id: ',  UDINT_TO_STRING(Errorid)));

	ELSIF MemFncAct = FNC_MOVE_REL
	THEN (* Relativ *)
		MCFctTxt											:= CONCAT('MC_MoveRelative TrigID No:',INT_TO_STRING(TrigID));
		Done 												:= MC_MoveRelative[TrigID].Done;
		Busy 												:= MC_MoveRelative[TrigID].Busy;
		Active 												:= MC_MoveRelative[TrigID].Active;
		CmdAborted 	 										:= MC_MoveRelative[TrigID].CommandAborted;
		Error												:=	MC_MoveRelative[TrigID].Error;
		ErrorId												:= MC_MoveRelative[TrigID].ErrorId;
		ErrorText											:= SEL(Error , '' ,  CONCAT('Error MC_MoveRelative id: ',  UDINT_TO_STRING(Errorid)));

	ELSIF MemFncAct = FNC_MOVE_ADD
	THEN (* Rel.Additive *)
		MCFctTxt											:= CONCAT('MC_MoveAdditive TrigID No:',INT_TO_STRING(TrigID));
		Done 												:= MC_MoveAdditive[TrigID].Done;
		Busy 												:= MC_MoveAdditive[TrigID].Busy;
		Active 												:= MC_MoveAdditive[TrigID].Active;
		CmdAborted 	 										:= MC_MoveAdditive[TrigID].CommandAborted;
		Error												:=	MC_MoveAdditive[TrigID].Error;
		ErrorId												:= MC_MoveAdditive[TrigID].ErrorId;
		ErrorText											:= SEL(Error , '' ,  CONCAT('Error MC_MoveAdditive id: ',  UDINT_TO_STRING(Errorid)));
		
	ELSIF MemFncAct = FNC_MOVE_VELO
	THEN (* Velocity *)
		MCFctTxt											:= CONCAT('MC_MoveVelo TrigID No:',INT_TO_STRING(TrigID));
		Active 												:= MC_MoveVelocity[TrigID].Active;
		Busy 												:= MC_MoveVelocity[TrigID].Busy ;
		CmdAborted 	 										:= MC_MoveVelocity[TrigID].CommandAborted;
		Error												:=	MC_MoveVelocity[TrigID].Error;
		ErrorId												:= MC_MoveVelocity[TrigID].ErrorId;
		ErrorText											:= SEL(Error , '' ,  CONCAT('Error MC_MoveVelocity id: ',  UDINT_TO_STRING(Errorid)));
		
	ELSIF MemFncAct > 0
	THEN
		MCFctTxt											:= CONCAT('Unknown Fnc no:', INT_TO_STRING(MemFncAct));
	ELSE                    							
		MCFctTxt											:= SEL(BusyIntern, 'NoAction' , 'Intern');
		Busy												:= BusyIntern;
		Done 												:= FALSE;
		Active 												:= FALSE;
		CmdAborted 											:= FALSE;
		Error												:=	FALSE;
		ErrorId												:= 0;
		ErrorText											:= '';
	END_IF

(* End funcktion *********************************************************************************)
	IF 	NOT rtExecuteMethod.CLK 
		AND NOT Busy 
		AND NOT Error 
		AND NOT Done 
		AND NOT Active 
		AND NOT CmdAborted
	THEN

		rtExecute(CLK := FALSE); 										
											
		IF MC_Jog.Busy
			OR MC_Halt.Busy
			OR MC_Stop.Busy
			OR MC_MoveVeloPreTrig.Busy
			OR MC_MoveAbsolute[1].Busy OR MC_MoveAbsolute[2].Busy
			OR MC_MoveModulo[1].Busy OR MC_MoveModulo[2].Busy
			OR MC_MoveRelative[1].Busy OR MC_MoveRelative[2].Busy 
			OR MC_MoveAdditive[1].Busy OR MC_MoveAdditive[2].Busy 
			OR MC_MoveVelocity[1].Busy OR MC_MoveVelocity[2].Busy 
		THEN (* Ablauffehler , es darf kein Baustein an dieser Stelle Busy sein *)
			MemFnc											:= -2;
		ELSE                								
			MemFnc											:= -1;
		END_IF              	
	END_IF

(**************************************************************************************************)
END_METHOD

METHOD PUBLIC Halt : BOOL //Result = Busy
//required parameter
//rAxis
//BufferMode
//Dec
//Jerk
//MoveOptions
VAR_INPUT
	Execute													:	BOOL;
END_VAR
MemFnc 														:= FNC_HALT;
THIS^.Execute												:= Execute;
_MCIntern();            									
Halt														:= Busy;
END_METHOD

METHOD PUBLIC JogOff : BOOL
VAR_INPUT
END_VAR
JogBwd 														:= JogFwd := FALSE;
IF __ISVALIDREF(rAxis)
THEN
	JogOff 													:= MemFnc = FNC_MOVE_JOG AND NOT rAxis.Status.Moving;
ELSE
	JogOff 													:= MemFnc = FNC_MOVE_JOG;
END_IF
END_METHOD

METHOD PUBLIC MoveAbs : BOOL //Result = Busy
//required parameter
//rAxis
//BufferMode
//Target
//Velo
//Acc
//Dec
//Jerk
//MoveOptions
VAR_INPUT
	Execute													:	BOOL;
END_VAR
MemFnc 														:= FNC_MOVE_ABS;
THIS^.Execute												:= Execute;
_MCIntern();            									
MoveAbs														:= Busy;
END_METHOD

METHOD PUBLIC MoveAdd : BOOL //Result = Busy
//required parameter
//rAxis
//BufferMode
//Target
//Velo
//Acc
//Dec
//Jerk
//MoveOptions
VAR_INPUT
	Execute													:	BOOL;
END_VAR
MemFnc 														:= FNC_MOVE_ADD;
THIS^.Execute												:= Execute;
_MCIntern();            									
MoveAdd														:= Busy;
END_METHOD

METHOD PUBLIC MoveJog : BOOL  //Result = Busy
//required parameter
//rAxis
//Direction
//JogMode	
//Target
//Velo
//Acc
//Dec
//Jerk
VAR_INPUT
	Execute													:	BOOL;
END_VAR
MemFnc 														:= FNC_MOVE_JOG;
THIS^.Execute												:= Execute;
_MCIntern();        										
MoveJog														:= Busy;
END_METHOD

METHOD PUBLIC MoveMod : BOOL //Result = Busy
//required parameter
//rAxis
//BufferMode
//Target
//Direction
//Velo
//Acc
//Dec
//Jerk
//MoveOptions
VAR_INPUT
	Execute													:	BOOL;
END_VAR
MemFnc 														:= FNC_MOVE_MOD;
THIS^.Execute												:= Execute;
_MCIntern();            									
MoveMod														:= Busy;
END_METHOD

METHOD MoveRel : BOOL //Result = Busy
//required parameter
//rAxis
//BufferMode
//Target
//Velo
//Acc
//Dec
//Jerk
//MoveOptions
VAR_INPUT
	Execute													:	BOOL;
END_VAR
MemFnc 														:= FNC_MOVE_REL;
THIS^.Execute												:= Execute;
_MCIntern();            									
MoveRel														:= Busy;
END_METHOD

METHOD PUBLIC MoveVelo : BOOL //Result = Busy
//required parameter
//rAxis
//BufferMode
//Direction
//Velo
//Acc
//Dec
//Jerk
//MoveOptions
VAR_INPUT
	Execute													:	BOOL;
END_VAR
MemFnc														:= FNC_MOVE_VELO;
THIS^.Execute												:= Execute;
_MCIntern();            									
MoveVelo													:= Busy;
END_METHOD

METHOD PUBLIC Stop : BOOL //Result = Busy
//required parameter
//rAxis
//Dec
//Jerk
//MoveOptions
VAR_INPUT
	Execute													:	BOOL;
END_VAR
MemFnc 														:= FNC_STOP;
THIS^.Execute												:= Execute;
_MCIntern();            									
Stop														:= busy;
END_METHOD

END_FUNCTION_BLOCK

// ---- POUs/PTP/02_Options/Drive/CanOpen/Ax_CanOpenDriveEventCtrl.TcPOU
FUNCTION_BLOCK Ax_CanOpenDriveEventCtrl
VAR CONSTANT
	CANTYPE_STAEUBLI										:	BOOL := FALSE;
END_VAR                             						
VAR_INPUT                           						
	EnableEvent												:	BOOL := TRUE;
	InAck													:	BOOL := FALSE; (* Reset Drive Flag *)
	Name													:	STRING(30) := '';
	ErrorEndlagePos											:	BOOL := FALSE;
	ErrorEndlageNeg											:	BOOL := FALSE;
	ErrorSchutzschalter										:	BOOL := FALSE;
	rAxis													:	REFERENCE TO AXIS_REF := 0; (* Pointer damit Aktionen Extern ohne Parameter aufgerufen werden können *)
END_VAR
VAR_IN_OUT
END_VAR
VAR_OUTPUT
	Busy													:	BOOL;
	Error													:	BOOL;
	ErrorId													:	UDINT;
	Fault													:	BOOL; (* Drive Error *)
	Ready													:	BOOL; (* Drive Ready *)
                                					
	LiveCountTimeout										:	BOOL;
	LiveCount										AT %I* 	:	USINT;	(* Wenn diese Variable nicht vorhanden ist bitte mit NCtoPLC *)


	RT_StatusChanged 										: BOOL;

	CanNodeSTATE									AT %I* 	:	USINT; (* Master- AND Slave-Mode:
   																						0 = No error
                        							
																						Master-Mode:
																						   1 = Node deactivated
																						   2 = Node not found
																						   4 = SDO syntax error at StartUp
																						   5 = SDO data mismatch at StartUp
																						   8 = Node StartUp in progress
																						  11 = FC510x Bus-OFF
																						  12 = Pre-Operational
																						  13 = Severe bus fault
																						  14 = Guarding: toggle error
																						  20 = TxPDO too short
																						  22 = Expected TxPDO is missing
																						  23 = Node is Operational but not all TxPDOs were received
																						  31 = only for EtherCAT gateways: WC-State of cyclic EtherCAT frame is 1
                        							
																						Slave-Mode:
																						 128 = Node is Operational but not all RxPDOs were received
																						 129 = Node is Pre-Operational
																						 130 = Node is Stopped *)
	EventStatusByte											:	BYTE;
END_VAR                             						
VAR_OUTPUT CONSTANT                 						
	SOURCE_DRIVES_CAN										:	UDINT := 1900;
END_VAR
VAR
END_VAR
VAR

(* Zwischenspeicher *********************************************************************)
	MemLiveCount											:	USINT;

	_StatusWord										AT %I* 	:	UINT;

	Status_Calibrated										:	BOOL;
	Status_FollowingError									:	BOOL;
	Status_TargetPosCntrLoop								:	BOOL;
	Status_InternalLimitActive								:	BOOL;
	Status_TargetReached									:	BOOL;
	Status_RemoteActiv										:	BOOL;
	Status_ManufacturerSpecific								:	BOOL;
	Status_Warning											:	BOOL;
	Status_SwitchOnDisabled									:	BOOL;
	Status_QuickStopNS										:	BOOL;
	Status_VoltageEnable									:	BOOL;
	Status_Fault											:	BOOL;
	Status_OperationEnabled									:	BOOL;
	Status_SwitchedOn										:	BOOL;
	Status_ReadyToSwitchOn									:	BOOL;
	Status_TxPDOToggle										:	BOOL;


(* Timer ********************************************************************************)
	TON_LiveCountTimeout									:	TON;
	TON_NotEnabled											:	TON;
                                    						
(* Trigger ******************************************************************************)

(* Bausteine ****************************************************************************)
	Event													:	EventClass25;

(* Dummy Speicher **********************************************************)
	i													: UINT := 0 ;

(****************************************************************************)
END_VAR

	(************************************************************************************)
	(*																					*)
	(*		B E C K H O F F   N E W   A U T O M A T I O N   T E C H N O L O G Y    		*)
	(*																					*)
	(*		Eiserstr.5	D-33415 Verl	Germany	phone:	+49-5246-0	www.Beckhoff.Com	*)
    (*																					*)
    (*		Bausteinbeschreibung	:	CanOpen Drive Ctrl								*)
	(*		TwinCAT-Version			:	2.1x		 									*)
	(*		Version					:	V1.2/ 04/13										*)
 	(*		Autor					:	JHUE/DS											*)
	(*		Lib						:													*)
	(*																					*)
	(************************************************************************************)

(* abort function-call if the reference is invalid *****************************)
IF NOT __ISVALIDREF(rAxis) 
THEN
	Busy													:= NOT Error;
	Fault													:= TRUE;
	Ready													:= FALSE;
	Error													:= TRUE;
	ErrorId													:= 16#4B30;
	RETURN;         										
END_IF

(* Read Statusword ********************************************************)
IF NOT CANTYPE_STAEUBLI
THEN
	Status_Calibrated										:= FALSE;
	Status_FollowingError									:= FALSE;
	Status_TargetPosCntrLoop								:= _Statusword.12;
	Status_InternalLimitActive								:= _Statusword.11;
	Status_TargetReached									:= FALSE;
	Status_TxPDOToggle										:= _Statusword.10; (* EL7201 *)
	Status_RemoteActiv										:= FALSE;
	Status_ManufacturerSpecific								:= FALSE;
	Status_Warning											:= _Statusword.7;
	Status_SwitchOnDisabled									:= _Statusword.6;
	Status_QuickStopNS										:= _Statusword.5;
	Status_VoltageEnable									:= FALSE;
	Status_Fault											:= _Statusword.3;
	Status_OperationEnabled									:= _Statusword.2;
	Status_SwitchedOn										:= _Statusword.1;
	Status_ReadyToSwitchOn									:= _Statusword.0;

	(* EL72xx DS402 Statusword
		Bit 0 : Ready to switch on
		Bit 1 : Switched on
		Bit 2 : Operation enabled
		Bit 3 : Fault
		Bit 4 : reserved
		Bit 5 : Quick stop (inverse)
		Bit 6 : Switch on disabled
		Bit 7 : Warning
		Bit 8 + 9 : reserved
		Bit 10 : TxPDOToggle (An-/Abwahl über 0x60DA)
		Bit 11 : Internal limit active
		Bit 12 : (Target value ignored)
		Bit 13 - 15 : reserved *)
ELSE
	(* LiveCount Timeout ************************************)
	TON_LiveCountTimeout(
		IN := MemLiveCount = LiveCount,
		PT := t#1s,
		Q	=> LiveCountTimeout);
	
	(* DriveStatusword *****************************)
	IF LiveCountTimeout 
	THEN 
		_StatusWord 										:= 0; 
	END_IF

	Status_Calibrated										:= _Statusword.14;
	Status_FollowingError									:= _Statusword.13;
	Status_TargetPosCntrLoop								:= _Statusword.12;
	Status_InternalLimitActive								:= _Statusword.11;
	Status_TargetReached									:= _Statusword.10;
	Status_TxPDOToggle										:= FALSE;
	Status_RemoteActiv										:= _Statusword.9;
	Status_ManufacturerSpecific								:= _Statusword.8;
	Status_Warning											:= _Statusword.7;
	Status_SwitchOnDisabled									:= _Statusword.6;
	Status_QuickStopNS										:= _Statusword.5;
	Status_VoltageEnable									:= _Statusword.4;
	Status_Fault											:= _Statusword.3;
	Status_OperationEnabled									:= _Statusword.2;
	Status_SwitchedOn										:= _Statusword.1;
	Status_ReadyToSwitchOn									:= _Statusword.0;
	(*
	Bits 	Value 	Description
	15		 X 		Reserved
	14 	0/1 		Status OF position feedback value.  1: the robot axis is calibrated.  0: the robot axis is NOT calibrated.
	13 	0/1 		No following error /Following error
	12 	0/1 		Target position ignored  /Target position shall be used as input TO position control loop
	11 	0/1 		Internal LIMIT active
	10 	0/1		Target reached
	9 		0/1 		Remote
	8 		0/1 		Manufacturer specific
	7 		0/1 		Warning
	6 		0/1 		Switch on disabled
	5 		1 			Quick stop. NS
	4 		0/1 		Voltage enable
	3 		0/1 		Fault
	2 		0/1 		Operation enabled
	1 		0/1 		Switched on
	0 		0/1 		Ready TO switch on
	*)

END_IF

(* DriveStatusBits ***********************************************)
	Fault													:= Status_Fault
																OR Status_FollowingError
																OR(NOT Status_Calibrated AND CANTYPE_STAEUBLI) (* Nur bei Absolut Encoder Achsen *)
																OR rAxis.NcToPlc.StateDWord.28 (* DriveDeviceError *)
																OR rAxis.NcToPlc.StateDWord.30; (* IODataInvalid *)
            												
	Ready 													:= NOT Fault
																	AND(Status_ReadyToSwitchOn OR Status_SwitchedOn);

(* Event Logger Meldungen *****************************************************)
	TON_NotEnabled(
		IN := Status_SwitchedOn AND NOT Status_OperationEnabled AND Ready,
		PT := t#2s);

	Event.no[1].Flag 										:= NOT Status_ReadyToSwitchOn; Event.no[1].Class := TC2_SYSTEM.TCEVENTCLASS_HINT;
	Event.no[2].Flag 										:= Status_FollowingError AND CANTYPE_STAEUBLI;
	Event.no[3].Flag 										:= Status_Fault;
	Event.no[4].Flag 										:= Status_Warning; 				Event.no[4].Class := TC2_SYSTEM.TCEVENTCLASS_WARNING;
	Event.no[5].Flag 										:= Status_InternalLimitActive;
	Event.no[6].Flag 										:= NOT Status_RemoteActiv AND CANTYPE_STAEUBLI;
	Event.no[7].Flag 										:= Status_SwitchOnDisabled;
	Event.no[8].Flag 										:= NOT Status_Calibrated AND CANTYPE_STAEUBLI; 	(* Nur bei Absolut Encoder Achsen *)
	Event.no[9].Flag 										:= Status_FollowingError AND CANTYPE_STAEUBLI;
	Event.no[10].Flag 										:= CanNodeSTATE = 128; 					(* Node is Operational but not all RxPDOs were received *)
	Event.no[11].Flag 										:= CanNodeSTATE = 129; 					(* Node is Pre-Operational *)
	Event.no[12].Flag 										:= CanNodeSTATE = 130;					(* Node is Stopped *)
	Event.no[13].Flag 										:= TON_NotEnabled.Q; 			Event.no[9].Class := TC2_SYSTEM.TCEVENTCLASS_WARNING;
	Event.no[14].Flag 										:= LiveCountTimeout AND CANTYPE_STAEUBLI; 			Event.no[10].Class := TC2_SYSTEM.TCEVENTCLASS_WARNING;
	Event.no[15].Flag 										:= ErrorSchutzschalter;
	Event.no[16].Flag 										:= ErrorEndlagePos;
	Event.no[17].Flag 										:= ErrorEndlageNeg;
	Event.no[18].Flag 										:= FALSE;
	Event.no[19].Flag 										:= FALSE;
	Event.no[20].Flag 										:= FALSE;
	Event.no[21].Flag 										:= FALSE;
	Event.no[22].Flag 										:= FALSE;
	Event.no[23].Flag 										:= FALSE;
	Event.no[24].Flag 										:= FALSE;
	Event.no[25].Flag 										:= FALSE;

(* Check if msg activ and init some parameter ***********************)
	IF Event.no[1].Text2 <> Name OR Event.no[1].Text2 <> ''
	THEN
		(* Init axisname *)
		FOR i := Event.MIN_EVENT TO Event.MAX_EVENT DO
		(*	Event.no[i].Text1								:= '';*)
			Event.no[i].Text2								:= SEL(LEN(name)>1,CONCAT('Axis id:',DWORD_TO_STRING(rAxis.NcToPlc.AxisId)),name);
		END_FOR
	END_IF

(* workl Event Ctrl *************************************************)
	Event(
		InAck 			:= InAck,
		Disable			:= rAxis.NcToPlc.AxisId = 0 OR NOT EnableEvent,
		SourceId		:= SOURCE_DRIVES_CAN + rAxis.NcToPlc.AxisId,
		
		StatusByte 		=> EventStatusByte);

(******************************************************************************)

METHOD PUBLIC Ack : bool
VAR_INPUT
END_VAR
Event.Ack();
END_METHOD

END_FUNCTION_BLOCK

// ---- POUs/EventLogger/TriggerEvents/EventClass25.TcPOU
{attribute 'no_check'}
FUNCTION_BLOCK EventClass25
VAR_OUTPUT CONSTANT
	MIN_EVENT												:	UINT := 1;
	MAX_EVENT												:	UINT := 25;
END_VAR                                                 	
VAR_INPUT                                               	
	InAck													:	BOOL := FALSE;
	SourceId												: 	UDINT := 0;
	no														:	ARRAY	[MIN_EVENT..MAX_EVENT] OF EventCtrl;
	Disable													:	BOOL := FALSE;
	AutoQuit												:	BOOL := FALSE; (* Ack error if flag is gone *)
	SetClass												:	E_TcEventClass := TC2_SYSTEM.TCEVENTCLASS_ALARM; (* if <> ALARM -> all Ctrls set dto this Eventclass *)
END_VAR                                                 	
VAR_OUTPUT                                              	
{attribute 'displaymode':='binary'}                     	
	StatusByte												:	BYTE := 0; //.0 HINT / .1 MSG / .2 ERR / .7 ACK
	CntEvents												:	UINT := 0; //Anzahl Events
END_VAR                                                 	
VAR                                                     	
	_Mem													:	BYTE;
	Disabled												:	BOOL;
	i 														:	UINT;
END_VAR

(* Eventclass 				V3.0	*)
(************************************)

(* status ***************************)
StatusByte := 0; CntEvents := 0;
IF(Disable OR SourceId = 0)AND Disabled
THEN
	RETURN;
ELSE
	Disabled												:= Disable OR SourceId = 0;
	                                                    	
FOR i := MIN_EVENT TO MAX_EVENT                         	
	DO                                                  	
		(* Init Default Class *)                        	
		IF 	SetClass <> TC2_SYSTEM.TCEVENTCLASS_ALARM   	
			AND NOT _Mem.7                              	
		THEN                                            	
			no[i].Class										:= SetClass;
			_Mem.7											:= i = MAX_EVENT;
		END_IF                                          			
		                                                			
		IF Disable OR SourceId = 0                      			
		THEN                                            			
			no[i].Flag 										:= FALSE;
			no[i].Quit 										:= no[i].State <> TCEVENTSTATE_INVALID AND no[i].State <> TCEVENTSTATE_RESETCON;
			Disabled										:= NOT no[i].Flag AND NOT no[i].Quit AND Disabled;
		ELSIF InAck                                     	
		THEN                                            	
			no[i].Quit 										:= TRUE;
			_Mem.0 											:= InAck;
                                                        	
		ELSIF _Mem.0                                    	
		THEN                                            	
			no[i].Quit 										:= FALSE;
			_Mem.0 											:= i <> MAX_EVENT;

		ELSIF AutoQuit
		THEN
			IF NOT no[i].Flag
				AND no[i].State <> TCEVENTSTATE_INVALID
				AND no[i].State <> TCEVENTSTATE_RESETCON
			THEN
				no[i].Quit 									:= TRUE;
			ELSE
				no[i].Quit 									:= FALSE;
			END_IF
		END_IF

		(* Mem current Event *)
		_Mem.1 := no[i].State <> TCEVENTSTATE_INVALID AND no[i].State <> TCEVENTSTATE_RESETCON;

		IF no[i].State <> TCEVENTSTATE_INVALID OR no[i].Flag THEN
			(* Call Event *)
			no[i](
				Flag	:= ,
				Quit	:= ,
				MsgId	:= i,
				SourceId:= SourceId,
				Class	:= (* see class call *),
				Text1	:= (* see class call *),
				Text2	:= (* see class call *),
				pText3	:= (* see class call *),
				State	=> );
		END_IF

		(* Set info flags *)
		IF no[i].State <> TCEVENTSTATE_INVALID AND no[i].State <> TCEVENTSTATE_RESETCON THEN
			CntEvents										:= CntEvents + 1;
			CASE no[i].Class OF                         	
			TC2_SYSTEM.TCEVENTCLASS_NONE,               	
			TC2_SYSTEM.TCEVENTCLASS_MESSAGE,            	
			TC2_SYSTEM.TCEVENTCLASS_HINT,               	
			TC2_SYSTEM.TCEVENTCLASS_STATEINFO,          	
			TC2_SYSTEM.TCEVENTCLASS_INSTRUCTION:        	
				StatusByte.0 								:= no[i].Flag OR no[i].state.0; (* Signaled *)
                                                        	
			TC2_SYSTEM.TCEVENTCLASS_WARNING,            	
			TC2_SYSTEM.TCEVENTCLASS_MAINTENANCE:        	
				StatusByte.7 								:= StatusByte.7 OR no[i].state.1; (* Gegangen *)
				StatusByte.1 								:= no[i].Flag OR no[i].state.0; (* Signaled *)
                                                        	
			TC2_SYSTEM.TCEVENTCLASS_ALARM,              	
			TC2_SYSTEM.TCEVENTCLASS_PARAMERROR:         	
				StatusByte.7 								:= StatusByte.7 OR no[i].state.1; (* Gegangen *)
				StatusByte.2 								:= no[i].Flag OR no[i].state.0; (* Signaled *)
                                                        	
			ELSE (* Unkown Class *)                     	
				StatusByte.2								:= TRUE;
                                                        	
			END_CASE

		ELSIF _Mem.1 
		THEN (* Send one time info event is gone *)
			; 
		ELSE
			; (* No error at this call *)
		END_IF


	END_FOR
	
END_IF
(********************************************)

METHOD PUBLIC Ack 
VAR_INPUT
END_VAR
FOR i := MIN_EVENT TO MAX_EVENT 
DO
	no[i](Quit := TRUE);
END_FOR

_Mem.0				:= TRUE;
END_METHOD

END_FUNCTION_BLOCK

// ---- POUs/EventLogger/TriggerEvents/EventCtrl.TcPOU
{attribute 'no_check'}
FUNCTION_BLOCK EventCtrl
VAR_INPUT
	Flag													:	BOOL := FALSE;
	Quit													:	BOOL := FALSE;
	MsgId													:	UINT := 0;
	SourceId												: 	UDINT:= 0;
	Class													:	E_TcEventClass := TC2_SYSTEM.TCEVENTCLASS_ALARM;
																				(*	TC2_SYSTEM.TCEVENTCLASS_NONE		-> QuitRequired = FALSE
																					TC2_SYSTEM.TCEVENTCLASS_MAINTENANCE-> QuitRequired = TRUE
																					TC2_SYSTEM.TCEVENTCLASS_MESSAGE		-> QuitRequired = FALSE
																					TC2_SYSTEM.TCEVENTCLASS_HINT		-> QuitRequired = FALSE
																					TC2_SYSTEM.TCEVENTCLASS_STATEINFO	-> QuitRequired = FALSE
																					TC2_SYSTEM.TCEVENTCLASS_INSTRUCTION	-> QuitRequired = FALSE
																					TC2_SYSTEM.TCEVENTCLASS_WARNING		-> QuitRequired = TRUE
																					TC2_SYSTEM.TCEVENTCLASS_ALARM		-> QuitRequired = TRUE
																					TC2_SYSTEM.TCEVENTCLASS_PARAMERROR	-> QuitRequired = TRUE *)

	Text1													:	STRING(20) := '';
	Text2													:	STRING(40) := '';
	pText3													:	POINTER TO STRING := 0; (* Pointer for special text *)
END_VAR
VAR_OUTPUT
	State													:	UDINT; (*	TCEVENTSTATE_INVALID  	: WORD := 16#0000; 		(* Invalid state some errors occured *)
																			TCEVENTSTATE_SIGNALED  	: WORD := 16#0001; 		(* The event is signaled *)
																			TCEVENTSTATE_RESET  	: WORD := 16#0002; 		(* The event is reset *)
																			TCEVENTSTATE_CONFIRMED  : WORD := 16#0010 (16); (* The event is confirmed *)
																			TCEVENTSTATE_RESETCON  	: WORD := 16#0012 (18); (* The event is reset and confirmed*)*)
END_VAR
VAR
	format													:	STRING(10) := '%s%s%s';
	pPara													:	ARRAY[1..3] OF PVOID;
	TmpString												:	STRING(1) := '';
	AdsEvent												:		ADSLOGEVENT :=(
																					NETID				:= '',
																					PORT				:= AMSPORT_EVENTLOG,
																					TMOUT 				:= DEFAULT_ADS_TIMEOUT,
																					EventConfigData 	:= (
																					Class 				:= TC2_SYSTEM.TCEVENTCLASS_ALARM,
																					Prio 				:= TCEVENTPRIO_IMPLICIT,
																					ProgId 				:= 'TcEventFormatter.TcXmlFormatter',
																					Flags 				:= 16#0140 (* TCEVENTFLAG_LOG OR TCEVENTFLAG_SRCID *),
																					StreamType 			:= TCEVENTSTREAM_SIMPLE (* TCEVENTSTREAM_NORMAL *),
																					bQuitRequired 		:= TRUE));
END_VAR

(* Event Ctrl-Meldung including textinfos which are send to the eventlogger V3.0 DS	*)
(* specific eventclasses have to be quit											*)
(************************************************************************************)

(* sequence *************************************************************)
	IF AdsEvent.Event
		OR State <> TCEVENTSTATE_INVALID
	THEN (* work EventLogger *)
		AdsEvent(
			NETID			:= ,(* see declaration *)
			PORT			:= ,(* see declaration *)
			Event			:= Flag OR AdsEvent.EventState = TCEVENTSTATE_INVALID AND NOT AdsEvent.Quit, (* Set Event until state <> invalid *)
			EventQuit		:= AdsEvent.EventState <> TCEVENTSTATE_INVALID
								AND AdsEvent.EventConfigData.bQuitRequired
								AND NOT AdsEvent.Eventstate.4
								AND NOT AdsEvent.Quit
								AND(
								Quit
								OR AdsEvent.EventQuit), (* quit send *)
			EventConfigData	:= ,(* see declaration *)
			EventDataAddress:= ADR(pPara),
			EventDataLength	:= 0,
			FbCleanup		:= NOT AdsEvent.FbCleanup AND AdsEvent.Err ,
			TMOUT			:= ,(* see declaration *)
			EventState		=> ,
			Err				=> ,
			ErrId			=> ,
			Quit			=> );

		IF AdsEvent.Event
			AND AdsEvent.EventState = TCEVENTSTATE_INVALID
		THEN
			State 											:= TCEVENTSTATE_SIGNALED;
		ELSIF AdsEvent.Quit
			AND AdsEvent.EventState = TCEVENTSTATE_INVALID
			AND AdsEvent.EventQuit
			OR 
			AdsEvent.FbCleanup		
		THEN
			State 											:= TCEVENTSTATE_RESETCON;
		ELSE
			State											:= AdsEvent.EventState ;
		END_IF

	ELSIF	Flag 
			AND SourceId > 0 
	THEN (* fire event *)
		(* Event Config *)
		IF class = TC2_SYSTEM.TCEVENTCLASS_NONE 				
		THEN
			AdsEvent.EventConfigData.bQuitRequired 			:= FALSE;
		ELSIF class = TC2_SYSTEM.TCEVENTCLASS_MAINTENANCE 
		THEN
			AdsEvent.EventConfigData.bQuitRequired 			:= TRUE;
		ELSIF class = TC2_SYSTEM.TCEVENTCLASS_MESSAGE 		
		THEN
			AdsEvent.EventConfigData.bQuitRequired 			:= FALSE;
		ELSIF class = TC2_SYSTEM.TCEVENTCLASS_HINT 			
		THEN
			AdsEvent.EventConfigData.bQuitRequired 			:= FALSE;
		ELSIF class = TC2_SYSTEM.TCEVENTCLASS_STATEINFO 	
		THEN
			AdsEvent.EventConfigData.bQuitRequired 			:= FALSE;
		ELSIF class = TC2_SYSTEM.TCEVENTCLASS_INSTRUCTION 
		THEN
			AdsEvent.EventConfigData.bQuitRequired 			:= FALSE;
		ELSIF class = TC2_SYSTEM.TCEVENTCLASS_WARNING 		
		THEN
			AdsEvent.EventConfigData.bQuitRequired 			:= TRUE;
		ELSIF class = TC2_SYSTEM.TCEVENTCLASS_ALARM 		
		THEN
			AdsEvent.EventConfigData.bQuitRequired 			:= TRUE;
		ELSIF class = TC2_SYSTEM.TCEVENTCLASS_PARAMERROR 	
		THEN
			AdsEvent.EventConfigData.bQuitRequired 			:= TRUE;
		ELSE
			AdsEvent.EventConfigData.bQuitRequired 			:= TRUE;
		END_IF
		
		AdsEvent.EventConfigData.DataFormatStrAddress		:= ADR(format);
		AdsEvent.EventConfigData.Id 						:= UINT_TO_UDINT(MsgID);
		AdsEvent.EventConfigData.SourceId 					:= SourceId;
		AdsEvent.EventConfigData.Class						:= Class;

		(* Data *)
		pPara[1] 											:= ADR(Text1);
		pPara[2] 											:= ADR(Text2);
		pPara[3] 											:= SEL(pText3 <> 0,ADR(TmpString) ,pText3);

		IF AdsEvent.Err 
		THEN
			AdsEvent(
				Event			:= FALSE,
				EventQuit 		:= FALSE,
				EventDataAddress:= ADR(pPara),
				FbCleanup		:= NOT AdsEvent.FbCleanup,
				EventState		=> );
				
		ELSE (* Fire Event *)
			AdsEvent( 	Event			:= FALSE,
						EventQuit 		:= FALSE, 
						FbCleanup 		:= FALSE, 
						EventDataAddress:= ADR(pPara));
						
			AdsEvent( 	Event 	:= TRUE);
			State 											:= TCEVENTSTATE_SIGNALED;
		END_IF
	ELSE
		; (* Wait for new flag *)
	END_IF

(**********************************************************************************)

END_FUNCTION_BLOCK

// ---- POUs/PTP/02_Options/ErrorNc/Ax_ErrorNCEventCtrl.TcPOU
{attribute 'no_check'}
FUNCTION_BLOCK Ax_ErrorNCEventCtrl
(* you can modify the block *)
(* dont forget to change then xml file and merge into then Eventlogger project	*)
(* See text below to create an xml file!!!! *)
VAR CONSTANT
	SOURCE_AXIS												:	UDINT := 1800; // + Axis Id
END_VAR                     								
VAR_INPUT                   								
	Enable													:	BOOL := TRUE; (* Show alarm message, warnings or hint. always reported !!! *)
	InAck													:	BOOL := FALSE;
	Name													:	STRING(30) := '';
	SourceId												:	UDINT := SOURCE_AXIS;
	AxErrorId												:	UDINT := 0;
	CmdAborted												:	INT := 0; 
	rAxis													:	REFERENCE TO AXIS_REF := 0;
END_VAR
VAR_OUTPUT
{attribute 'displaymode':='binary'}
	StatusByte												:	BYTE;
	CntEvents												:	UINT;
END_VAR
VAR
(* Zwischenspeicher ***********************************************)
	QuitInternal 											: BOOL;

(* Timer **********************************************************)

(* Trigger ********************************************************)

(* Bausteine ******************************************************)
	Event													:	EventClass10 := (
																	AutoQuit				:= FALSE, 
																	SetClass 			:= TC2_SYSTEM.TCEVENTCLASS_ALARM );
	EventMsgCtrl											:	Ax_ErrorNCEventMsgCtrl;

(* Dummy Speicher *************************************************)
	i														:	UINT ;

END_VAR
(* Plc Ax Message template:
	Copy the text to any txt file an change the filetyp to .xml .
	Be sure that the xml file is already in the EventLogger project,
	after that, copy the new xml file into the "TcEventMessage.ecp Files" folder.

<TcEventSources>
	<Source>
		<Id>1800</Id>
		<Id>1801</Id>
		<Id>1802</Id>
		<Id>1803</Id>
		<Id>1804</Id>
		<Id>1805</Id>
		<Id>1806</Id>
		<Id>1807</Id>
		<Id>1808</Id>
		<Id>1809</Id>
		<Id>1810</Id>
		<Id>1811</Id>
		<Id>1812</Id>
		<Id>1813</Id>
		<Id>1814</Id>
		<Id>1815</Id>
		<Id>1816</Id>
		<Id>1817</Id>
		<Id>1818</Id>
		<Id>1819</Id>
		<Id>1820</Id>
		<Id>1821</Id>
		<Id>1822</Id>
		<Id>1823</Id>
		<Id>1824</Id>
		<Id>1825</Id>		
		<Id>1826</Id>
		<Id>1827</Id>
		<Id>1828</Id>
		<Id>1829</Id>
		<Id>1830</Id>
		<Name LcId="1031">Plc Axis Message</Name>
		<Name LcId="1033">Plc Axis Message</Name>
		<Event>
			<Id>1</Id>
			<ReqMustCon>0</ReqMustCon>
			<Message LcId="1031">%1 - NC-Störung IO Kommunikation zum Antrieb %2%3</Message>
			<Class>6</Class>
			<Priority>0</Priority>
		</Event>
		<Event>
			<Id>2</Id>
			<ReqMustCon>0</ReqMustCon>
			<Message LcId="1031">%1 - NC-Störung Antrieb %2%3</Message>
			<Class>6</Class>
			<Priority>0</Priority>
		</Event>
		<Event>
			<Id>3</Id>
			<ReqMustCon>0</ReqMustCon>
			<Message LcId="1031">%1 - Referenzfahrt aktiv %2%3</Message>
			<Class>6</Class>
			<Priority>0</Priority>
		</Event>
		<Event>
			<Id>4</Id>
			<ReqMustCon>0</ReqMustCon>
			<Message LcId="1031">%1 - Free %2%3</Message>
			<Class>6</Class>
			<Priority>0</Priority>
		</Event>
		<Event>
			<Id>5</Id>
			<ReqMustCon>0</ReqMustCon>
			<Message LcId="1031">%1 - Free %2%3</Message>
			<Class>6</Class>
			<Priority>0</Priority>
		</Event>
		<Event>
			<Id>6</Id>
			<ReqMustCon>0</ReqMustCon>
			<Message LcId="1031">%1 - Free %2 %3</Message>
			<Class>6</Class>
			<Priority>0</Priority>
		</Event>
		<Event>
			<Id>7</Id>
			<ReqMustCon>0</ReqMustCon>
			<Message LcId="1031">%1 - Free %2%3</Message>
			<Class>6</Class>
			<Priority>0</Priority>
		</Event>
		<Event>
			<Id>8</Id>
			<ReqMustCon>0</ReqMustCon>
			<Message LcId="1031">%1 - Free %2%3</Message>
			<Class>6</Class>
			<Priority>0</Priority>
		</Event>
		<Event>
			<Id>9</Id>
			<ReqMustCon>0</ReqMustCon>
			<Message LcId="1031">%1 - Free %2%3</Message>
			<Class>6</Class>
			<Priority>0</Priority>
		</Event>
		<Event>
			<Id>10</Id>
			<ReqMustCon>0</ReqMustCon>
			<Message LcId="1031">%1 - Free %2%3</Message>
			<Class>6</Class>
			<Priority>0</Priority>
		</Event>
		<Event>
			<Id>201</Id>
			<ReqMustCon>0</ReqMustCon>
			<Message LcId="1031">%1 %2 %3 @V1:%4 %5 @V2:%6</Message>
			<Class>6</Class>
			<Priority>0</Priority>
		</Event>
	</Source>
</TcEventSources>

*)

(* Error message axis to EventLogger 			V3.0	DS	*)
(***********************************************************)

(* Sequence **************************************************************)
IF __ISVALIDREF(rAxis) AND SourceId > 0 
THEN
	(* get Quit signal **************************************************)
	IF InAck 
	THEN 
		QuitInternal := TRUE; 
	END_IF (* set false see below *)

(* Event Logger Meldungen *****************************************************)
	Event.no[1].Flag 										:= rAxis.Status.IoDataInvalid;
	Event.no[2].Flag 										:= rAxis.Status.DriveDeviceError;
	Event.no[3].Flag 										:= rAxis.Status.Homing;   
	Event.no[4].Flag 										:= CmdAborted <> 0;  
	
	IF Event.no[4].Flag 
	THEN 
		Event.no[4].Text1 									:= INT_TO_STRING(CmdAborted);  
	END_IF
		Event.no[5].Flag 									:= FALSE;
		Event.no[6].Flag 									:= FALSE;
		Event.no[7].Flag 									:= FALSE;
		Event.no[8].Flag 									:= FALSE;
		Event.no[9].Flag 									:= FALSE;
		Event.no[10].Flag 									:= FALSE;

(* workl Event Ctrl *************************************************)
	IF Event.no[1].Text2 <> Name OR Event.no[1].Text2 <> ''
	THEN
		//Init EventClass
		Event.no[3].Class 									:= TC2_SYSTEM.TCEVENTCLASS_HINT;
		Event.no[4].Class 									:= TC2_SYSTEM.TCEVENTCLASS_WARNING;

		(* Init Name *)
		FOR i := Event.MIN_EVENT TO Event.MAX_EVENT DO
			Event.no[i].Text2								:= SEL(LEN(name)>1,CONCAT('Axis id:',DWORD_TO_STRING(rAxis.NcToPlc.AxisId)),name);
		END_FOR
	END_IF


	Event(
		InAck 		:= InAck,
		Disable		:= NOT Enable,
		SourceId	:= SourceId + rAxis.NcToPlc.AxisId,

		StatusByte 	=> StatusByte,
		CntEvents	=> );	

(* Send ErrorId Message Text **********************************)
	EventMsgCtrl(
		InAck		:= NOT Enable OR QuitInternal OR AxErrorId = 0 AND EventMsgCtrl.State <> 0,
		Name		:= name,
		AxId		:= rAxis.NcToPlc.AxisId,
		Flag		:= AxErrorId > 0 AND Enable,
		AxErrorID	:= AxErrorId,
		State		=> );

	StatusByte.2											:= StatusByte.2 OR EventMsgCtrl.State.0 ;
	StatusByte.7											:= StatusByte.7 OR EventMsgCtrl.State.1 ;
	CntEvents												:= SEL(EventMsgCtrl.State.2, CntEvents , CntEvents + 1); 
	
(* Error unkonw pointer or axis id *****************************)
ELSE
	EventMsgCtrl(Flag := FALSE, InAck := EventMsgCtrl.State <> 0);
	Event(Disable := TRUE, StatusByte => StatusByte , CntEvents => CntEvents);
END_IF

(* Default reset Quit Internal *******************************)
	QuitInternal 											:= FALSE;

(**************************************************************)

METHOD PUBLIC Ack : bool
VAR_INPUT
END_VAR
QuitInternal 												:= TRUE;
END_METHOD

END_FUNCTION_BLOCK

// ---- POUs/Lib/FB_HydLinearRamp.TcPOU
FUNCTION_BLOCK FB_HydLinearRamp
VAR_INPUT
	Enable		: BOOL;
	TargetSpeed	: REAL;
	AccStep		: REAL;
	DecStep		: REAL;
	MinOutput	: REAL;
	MaxOutput	: REAL;
END_VAR
VAR_OUTPUT
	CmdSpeed	: REAL;
	DoneToTarget: BOOL;
END_VAR
VAR
	rAbsCmd			: REAL;
	rAbsTarget		: REAL;
	rEffectiveTarget: REAL;
	rStep			: REAL;
	rLimitMax		: REAL;
	rLimitMin		: REAL;
END_VAR

rLimitMax	:= ABS(MaxOutput);
rLimitMin	:= ABS(MinOutput);

IF NOT Enable THEN
	CmdSpeed	:= 0.0;
	DoneToTarget:= TRUE;
ELSE
	rEffectiveTarget	:= LIMIT(-rLimitMax, TargetSpeed, rLimitMax);
	IF (ABS(rEffectiveTarget) > 0.0) AND (ABS(rEffectiveTarget) < rLimitMin) THEN
		rEffectiveTarget	:= SEL(rEffectiveTarget >= 0.0, -rLimitMin, rLimitMin);
	END_IF

	IF CmdSpeed * rEffectiveTarget < 0.0 THEN
		rEffectiveTarget	:= 0.0;
	END_IF

	rAbsCmd		:= ABS(CmdSpeed);
	rAbsTarget	:= ABS(rEffectiveTarget);

	IF rAbsTarget > rAbsCmd THEN
		rStep	:= ABS(AccStep);
	ELSE
		rStep	:= ABS(DecStep);
	END_IF

	IF rStep <= 0.0 THEN
		rAbsCmd	:= rAbsTarget;
	ELSIF rAbsTarget > rAbsCmd THEN
		IF (rAbsCmd < rLimitMin) AND (rAbsTarget > 0.0) THEN
			rAbsCmd	:= rLimitMin;
		END_IF
		rAbsCmd	:= MIN(rAbsCmd + rStep, rAbsTarget);
	ELSE
		rAbsCmd	:= MAX(rAbsCmd - rStep, rAbsTarget);
	END_IF

	IF rAbsCmd <= 0.0001 THEN
		CmdSpeed := 0.0;
	ELSIF rEffectiveTarget >= 0.0 THEN
		CmdSpeed := rAbsCmd;
	ELSE
		CmdSpeed := -rAbsCmd;
	END_IF

	DoneToTarget := ABS(CmdSpeed - rEffectiveTarget) <= 0.0001;
END_IF

END_FUNCTION_BLOCK

// ---- POUs/PTP/02_Options/Drive/Ethercat/Ax_EcMC2DriveCtrl.TcPOU
FUNCTION_BLOCK Ax_EcMC2DriveCtrl (* Lips: TcMc2Drive, TcDrive *)
VAR_INPUT
	RST														:	BOOL := FALSE; (* Reset Drive Flag *)
	SetReferenz												: 	BOOL := FALSE;
	Referenzpos												: 	LREAL := 0.0;
	rAxis													:	REFERENCE TO AXIS_REF := 0; (* Pointer damit Aktionen Extern ohne Parameter aufgerufen werden können *)
END_VAR                                 					
VAR_IN_OUT                              					
END_VAR                                 					
VAR_OUTPUT                              					
	Busy													:	BOOL;
	Error													:	BOOL;
	ErrorId													:	UDINT;
	SercosErrorId											:	UINT;
	ErrorText												:	STRING(40);
                                        					
	Fault													:	BOOL; (* Drive Error *)
	Ready													:	BOOL; (* Drive Ready *)
	InReferenz												:	BOOL; (* Drive in reference *)
                                    						
	Status													:	ST_AX5000DriveStatus;
	C1D														:	ST_AX5000_C1D;

	RT_StatusChanged	 									: BOOL;
	StatusWord										AT %I* 	: WORD; (* S-0-0135 - muss unter EA -> Ax5000 -> AT -> "DriveStatusWord" direkt verknüpft werden *)
	Operational												: INPUT := (Force := TRUE);	(* Betriebsbereit *)
	EcState											AT %I* 	: 	UINT; (* Ethercat InfoData State *)
END_VAR                  						
VAR_OUTPUT CONSTANT
END_VAR
VAR (* EA Internal *)
	_AmsNetId										AT %I*	:	ST_AmsAddr; (* Drive AMS Net Adr. *)
	_EcInfoDataState								AT %I* 	: 	UINT; (* Ethercat InfoData State *)
END_VAR
VAR

(* Zwischenspeicher *********************************************************************)

	_MemDriveStatusword										: 	WORD;
	_word													:	WORD;
	_DWORD													:	DWORD;
	MEM_StatusTrig											:	BYTE;
	StatusTrig												:	BYTE;
	stateReadStatus											:	INT;
	stateCtrl												:	INT := 0;

(* Timer ********************************************************************************)

(* Trigger ******************************************************************************)

(* Bausteine ****************************************************************************)
	SoEDriveReset											: 	FB_SoEReset;
	SoEWrite												: 	FB_SoEWrite;
	SoERead													: 	FB_SoERead;
	SoEExecuteCmd											:	FB_SoEExecuteCommand;
	EcSetSlaveSTATE											:	FB_EcSetSlaveSTATE;

(* Dummy Speicher **********************************************************)
	i														: 	INT := 0 ;

(****************************************************************************)
END_VAR

	(************************************************************************************)
	(*																					*)
	(*		B E C K H O F F   N E W   A U T O M A T I O N   T E C H N O L O G Y    		*)
	(*																					*)
	(*		Eiserstr.5	D-33415 Verl	Germany	phone:	+49-5246-0	www.Beckhoff.Com	*)
    (*																					*)
    (*		Bausteinbeschreibung	:	Ethercat MC2 Drive Ctrl							*)
	(*		TwinCAT-Version			:	3.x or higher	 								*)
	(*		Version					:	V3.0/05/11										*)
 	(*		Autor					:	Daniel Schlingmann								*)
	(*		Lib						:	TcMC2Drive.lib / TcDrive.Lib					*)
	(*																					*)
	(* Call cyclic																		*)
	(************************************************************************************)

(* abort function-call if the reference is invalid *****************************)
IF NOT __ISVALIDREF(rAxis)  
THEN
	Busy													:= NOT Error;
	Fault													:= TRUE;
	Ready													:= FALSE;
	Error													:= TRUE;
	ErrorId													:= 16#4B30;
	ErrorText												:= 'Referenz rAxis hat ungueltigen Wert(0)';
	SercosErrorId											:= 0;
	RETURN;
END_IF

(* DriveStatusword *****************************)
	Status 													:= F_ConvWordToSTAX5000DriveStatus(StatusWord);

(* Drive Operation Input ***********************)
	Operational(
		Force		:= ,
		Invert		:= ,
		PT_ON		:= ,
		PT_OFF		:= ,
		Q_DIRECT	=> ,
		Q			=> ,
		Q_RT		=> ,
		Q_FT		=> ,
		INPUT		=> );

(* DriveStatusBits ***********************************************)
	Fault													:= Status.bDrvShutdownBitC1D
																OR rAxis.NcToPlc.StateDWord.28 (* DriveDeviceError *)
																OR rAxis.NcToPlc.StateDWord.30; (* IODataInvalid *)
                                						
	Ready 													:= NOT Fault
																	AND(Status.bReadyForEnable OR Status.bEnabled)
																	AND Operational.Q;
                                	
(* Reset Drive ****************************************************)
	SoEDriveReset(
		NetId		:= ,
		Execute		:= ,
		Timeout		:= ,
		Axis		:= rAxis,
		Busy		=> ,
		Error		=> ,
		AdsErrId	=> ,
		SercosErrId	=> );

	IF SoEDriveReset.Busy 
	THEN
		; (* Block ist currend working *)
	ELSIF RST
	THEN
		Reset();
	ELSIF SoEDriveReset.Execute
	THEN
	(*	RefreshStatus(); *)
		SoEDriveReset.Execute := FALSE;
	END_IF

(* Set Etehrcat State to OP ********************************************)
	EcSetSlaveSTATE(
		sNetId		:= F_CreateAmsNetId(nIds := _AmsNetId.netId),
		nSlaveAddr	:= _AmsNetId.port,
		bExecute	:= ,
		tTimeout	:= DEFAULT_ADS_TIMEOUT,
		reqState	:= Tc2_EtherCAT.EC_DEVICE_STATE_OP,
		bBusy		=> ,
		bError		=> ,
		nErrId		=> ,
		currState	=> );

	IF EcSetSlaveSTATE.bBusy
	THEN
		; (* Block ist currend working *)
	ELSIF EcSetSlaveSTATE.bExecute
		AND NOT RST
	THEN
		RefreshStatus();
		EcSetSlaveSTATE.bExecute 							:= FALSE;
	END_IF

(* Referenzieren *******************************************************)
	CASE stateCtrl OF
	-1,0:
		IF SetReferenz
		THEN
			Referenz();
		ELSE
			stateCtrl										:= 0;
		END_IF

	1: (* Referezwert schreiben **************************************)
		IF NOT SoEWrite.Busy
			AND SoEWrite.Execute
		THEN
			IF SoEWrite.Error
			THEN
				stateCtrl 									:= 0;
			ELSE                							
				stateCtrl									:= 2;
			END_IF
		END_IF

		_DWORD := LREAL_TO_UDINT(Referenzpos);

		SoEWrite(
			NetId		:= ,
			Idn			:= S_0_IDN + 52,
			Element		:= EC_SOE_ELEMENT_VALUE ,
			pSrcBuf		:= ADR(_DWORD),
			BufLen		:= SIZEOF(_DWORD),
			Execute		:= stateCtrl = 1,
			Timeout		:= DEFAULT_ADS_TIMEOUT,
			Password	:= ,
			Axis		:= rAxis,
			Busy		=> ,
			Error		=> ,
			AdsErrId	=> ,
			SercosErrId	=> );

	2: (* commad for setting setvalue *)
		IF NOT SoEExecuteCmd.Busy
			AND SoEExecuteCmd.Execute
		THEN
			IF SoEExecuteCmd.Error
			THEN
				stateCtrl 									:= 0;
			ELSE
				RefreshStatus();
				IF NOT SetReferenz
				THEN
					stateCtrl 								:= 0;
				ELSE            							
					stateCtrl 								:= -1;
				END_IF
			END_IF
		END_IF

		SoEExecuteCmd(
			NetId		:= '',
			Idn			:= P_0_IDN + 12,
			Execute		:= stateCtrl = 2,
			Timeout		:= DEFAULT_ADS_TIMEOUT,
			Axis		:= rAxis,
			Busy		=> ,
			Error		=> ,
			AdsErrId	=> ,
			SercosErrId	=> );
	ELSE
		;
	END_CASE


(* evaluate sercos DriveStatusword *********************************************************)
	RT_StatusChanged 										:= SHR(Statusword,2) <> _MemDriveStatusword;
	_MemDriveStatusword 									:= SHR(Statusword,2);

(* Start Read Drive status *****************************************************************)
	CASE stateReadStatus OF
	0:
		StatusTrig.0 										:= rAxis.NcToPlc.StateDWord.28; (* DriveDeviceError *)
		StatusTrig.1 										:= rAxis.NcToPlc.StateDWord.30; (* IODataInvalid *)
                                							
		IF RT_StatusChanged
			OR MEM_StatusTrig <> StatusTrig
		THEN
			RefreshStatus();
		ELSE
			;
		END_IF

	(* Read Class 1 Diag *********************************************************)
	10:
		IF NOT SoERead.Busy
			AND SoERead.Execute
		THEN
			IF SoERead.Error
			THEN
				stateReadStatus 							:= 0;
			ELSE                    						
				C1D 										:= F_ConvWordToSTAX5000C1D(_word);
				stateReadStatus 							:= stateReadStatus + 1;
			END_IF
		END_IF

		SoERead(
			NetId		:= ,
			Idn			:= S_0_IDN + 11,
			Element		:= EC_SOE_ELEMENT_VALUE,
			pDstBuf		:= ADR(_word),
			BufLen		:= SIZEOF(_word),
			Execute		:= stateReadStatus = 10,
			Timeout		:= DEFAULT_ADS_TIMEOUT,
			Axis		:= rAxis,
			Busy		=> ,
			Error		=> ,
			AdsErrId	=> ,
			SercosErrId	=> ,
			Attribute	=> );

	(* S-0-0403 In Referenz ********************************************************)
	11:
		IF NOT SoERead.Busy
			AND SoERead.Execute
		THEN
			IF SoERead.Error
			THEN
				stateReadStatus 							:= 0;
			ELSE
				InReferenz 									:= _WORD.0 AND _WORD.1;
				stateReadStatus 							:= 0;
			END_IF
		END_IF

		SoERead(
			NetId		:= ,
			Idn			:= S_0_IDN + 403,
			Element		:= EC_SOE_ELEMENT_VALUE,
			pDstBuf		:= ADR(_word),
			BufLen		:= SIZEOF(_word),
			Execute		:= stateReadStatus = 11,
			Timeout		:= DEFAULT_ADS_TIMEOUT,
			Axis		:= rAxis,
			Busy		=> ,
			Error		=> ,
			AdsErrId	=> ,
			SercosErrId	=> ,
			Attribute	=> );

	(* reading status finished ************************************************************)
	ELSE (* Case else *)
		stateReadStatus 									:= 0;
	END_CASE

(* Error Hdl FB ******************************************************************)
	IF SoEDriveReset.Error
	THEN
		Error												:=	TRUE;
		ErrorId												:= 0;
		SercosErrorId										:= SoEDriveReset.SercosErrId;
		ErrorText											:= CONCAT('SoeDrvReset SercosErrId: ',DWORD_TO_HEXSTR(SoEDriveReset.SercosErrId,4,FALSE));
		ErrorText											:=	CONCAT(CONCAT(ErrorText,', ADSErrId: '),UINT_TO_STRING(SoEDriveReset.AdsErrId));
	ELSIF SoEExecuteCmd.Error
	THEN
		Error												:=	TRUE;
		ErrorId												:= 0;
		SercosErrorId										:= SoEExecuteCmd.SercosErrId;
		ErrorText											:= CONCAT('SoEExecuteCmd SercosErrId: ',DWORD_TO_HEXSTR(SoEExecuteCmd.SercosErrId,4,FALSE));
		ErrorText											:=	CONCAT(CONCAT(ErrorText,', ADSErrId: '),UINT_TO_STRING(SoEExecuteCmd.AdsErrId));
	ELSIF SoERead.Error
	THEN
		Error												:=	TRUE;
		ErrorId												:= 0;
		SercosErrorId										:= SoERead.SercosErrId;
		ErrorText											:= CONCAT('SoERead SercosErrId: ',DWORD_TO_HEXSTR(SoERead.SercosErrId,4,FALSE));
		ErrorText											:=	CONCAT(CONCAT(ErrorText,', ADSErrId: '),UINT_TO_STRING(SoERead.AdsErrId));
	ELSIF SoEWrite.Error
	THEN
		Error												:=	TRUE;
		ErrorId												:= 0;
		SercosErrorId										:= SoEWrite.SercosErrId;
		ErrorText											:= CONCAT('SoEWrite SercosErrId: ',DWORD_TO_HEXSTR(SoEWrite.SercosErrId,4,FALSE));
		ErrorText											:=	CONCAT(CONCAT(ErrorText,', ADSErrId: '),UINT_TO_STRING(SoEWrite.AdsErrId));
	END_IF

(* FB is Busy *******************************************************************)
	Busy 													:= stateCtrl > 0
																OR SoEDriveReset.Busy
																OR stateReadStatus > 0;

(******************************************************************************)

METHOD PUBLIC Referenz : BOOL //Result = Busy
VAR_INPUT
END_VAR
IF NOT __ISVALIDREF(rAxis)  
THEN
	Busy													:= NOT Error;
	Error													:= TRUE;
	ErrorId													:= 16#4B30;
	ErrorText												:= 'Referenz rAxis hat ungueltigen Wert(0)';
	SercosErrorId											:= 0;
ELSIF stateCtrl = 0 
THEN
	ErrorText												:= '';
	Error													:=	FALSE;
	ErrorId													:= 0;
	SercosErrorId											:= 0;
	Busy													:= TRUE;
	stateCtrl 												:= 1;
	SoEWrite(Execute := FALSE, Axis := rAxis);
	SoEExecuteCmd(Execute := FALSE, Axis := rAxis);
ELSE
	Busy													:= TRUE;
END_IF                              						
                                    	
Referenz													:= Busy;
END_METHOD

METHOD PUBLIC RefreshStatus : BOOL //Result = Busy
VAR_INPUT
END_VAR
IF NOT __ISVALIDREF(rAxis)  
THEN
	Busy													:= NOT Error;
	Error													:= TRUE;
	ErrorId													:= 16#4B30;
	ErrorText												:= 'Referenz rAxis hat ungueltigen Wert(0)';
	SercosErrorId											:= 0;
ELSIF stateReadStatus = 0 
THEN
	Busy													:= TRUE;
	Error													:= FALSE;
	ErrorTExt												:= '';
	ErrorId													:= 0;
	SercosErrorId											:= 0;
	stateReadStatus 										:= 10;
	StatusTrig.0 											:= rAxis.NcToPlc.StateDWord.28; (* DriveDeviceError *)
	StatusTrig.1 											:= rAxis.NcToPlc.StateDWord.30; (* IODataInvalid *)
	MEM_StatusTrig 											:= StatusTrig;
	SoERead(
		Execute := FALSE,
		Axis 	:= rAxis);
ELSE
	Busy													:= TRUE;
END_IF                              						
                                    						
RefreshStatus												:= Busy;
END_METHOD

METHOD PUBLIC Reset : BOOL //Result = Busy
VAR_INPUT
END_VAR
IF NOT SoEDriveReset.Execute
THEN
	Error													:=	FALSE;
	ErrorId													:= 0;
	SercosErrorId											:= 0;
	Errortext												:= '';
	Busy													:= TRUE;
	Reset													:= TRUE;
ELSE
	SoEDriveReset.Execute									:= TRUE;
	EcSetSlaveSTATE.bExecute								:= NOT (( UINT_TO_WORD(EcState) AND Tc2_EtherCAT.EC_DEVICE_STATE_MASK ) = Tc2_EtherCAT.EC_DEVICE_STATE_OP)
																AND EcState > 0;
											
	Reset													:= SoEDriveReset.Busy;				
END_IF
END_METHOD

END_FUNCTION_BLOCK

// ---- POUs/PTP/02_Options/Drive/Stepper/Ax_StepperDriveEventCtrl.TcPOU
FUNCTION_BLOCK Ax_StepperDriveEventCtrl
VAR CONSTANT
END_VAR
VAR_INPUT
	EnableEvent												:	BOOL := TRUE;
	InAck													:	BOOL := FALSE; (* Reset Drive Flag *)
	Name													:	STRING(30) := '';
	ErrorEndlagePos											:	BOOL := FALSE;
	ErrorEndlageNeg											:	BOOL := FALSE;
	ErrorSchutzschalter										:	BOOL := FALSE;
	rAxis													:	REFERENCE TO AXIS_REF := 0; (* Pointer damit Aktionen Extern ohne Parameter aufgerufen werden können *)
END_VAR                     					
VAR_IN_OUT                  					
END_VAR                     					
VAR_OUTPUT                  					
	Busy													:	BOOL;
	Error													:	BOOL;
	ErrorId													:	UDINT;
	Fault													:	BOOL; (* Drive Error *)
	Ready													:	BOOL; (* Drive Ready *)
                            					
	RT_StatusChanged 										: 	BOOL;
	EventStatusByte											:	BYTE;
END_VAR                     					
VAR_OUTPUT CONSTANT         	
	SOURCE_DRIVES_STEPPER									:	UDINT := 1600;
END_VAR                     					
VAR                         					
	_StatusWord										AT %I* 	:	UINT;
                            	
END_VAR
VAR

(* Zwischenspeicher *********************************************************************)
	Status_ReadyToEnable									: BOOL;
	Status_Ready											: BOOL;
	Status_Warning											: BOOL;
	Status_Error											: BOOL;
	Status_MovingPos										: BOOL;
	Status_MovingNeg										: BOOL;
	Status_TorqueReduced									: BOOL;
	Status_MotorStall										: BOOL;
	Status_DigInput1										: BOOL;
	Status_DigInput2										: BOOL;
	Status_SyncError										: BOOL;
	Status_TxPDOToggle										: BOOL;


(* Timer ********************************************************************************)
	TON_LiveCountTimeout									:	TON;
	TON_NotEnabled											:	TON;

(* Trigger ******************************************************************************)

(* Bausteine ****************************************************************************)
	Event													:	EventClass10;

(* Dummy Speicher **********************************************************)
	i														: UINT := 0 ;

(****************************************************************************)
END_VAR

	(************************************************************************************)
	(*																					*)
	(*		B E C K H O F F   N E W   A U T O M A T I O N   T E C H N O L O G Y    		*)
	(*																					*)
	(*		Eiserstr.5	D-33415 Verl	Germany	phone:	+49-5246-0	www.Beckhoff.Com	*)
    (*																					*)
    (*		Bausteinbeschreibung	:	Stepper Drive ctrl								*)
	(*		TwinCAT-Version			:	2.1x		 									*)
	(*		Version					:	V1.2/ 04/13										*)
 	(*		Autor					:	JHUE/DS											*)
	(*		Lib						:													*)
	(*																					*)
	(************************************************************************************)

(* abort function-call if the reference is invalid *****************************)
IF NOT __ISVALIDREF(rAxis) 
THEN
	Busy													:= NOT Error;
	Fault													:= TRUE;
	Ready													:= FALSE;
	Error													:= TRUE;
	ErrorId													:= 16#4B30;
	RETURN;
END_IF

(* Read Statusword ********************************************************)
	Status_ReadyToEnable									:= _StatusWord.0;
	Status_Ready											:= _StatusWord.1;
	Status_Warning											:= _StatusWord.2;
	Status_Error											:= _StatusWord.3;
	Status_MovingPos										:= _StatusWord.4;
	Status_MovingNeg										:= _StatusWord.5;
	Status_TorqueReduced									:= _StatusWord.6;
	Status_MotorStall										:= _StatusWord.7;
//	_StatusWord.8; //0                  					
//	_StatusWord.9; //1                  					
//	_StatusWord.10;//2                  					
	Status_DigInput1										:= _StatusWord.11;
	Status_DigInput2										:= _StatusWord.12;
	Status_SyncError										:= _StatusWord.13;
//	_StatusWord.14;//6
	Status_TxPDOToggle										:= _StatusWord.15;
	
(* DriveStatusBits ***********************************************)
	Fault													:= Status_Error
															//	OR Status_MotorStall
																OR Status_SyncError
																OR rAxis.NcToPlc.StateDWord.28 (* DriveDeviceError *)
																OR rAxis.NcToPlc.StateDWord.30; (* IODataInvalid *)
         											
	Ready	 												:= NOT Fault
																AND(Status_ReadyToEnable OR Status_Ready);

(* Event Logger Meldungen *****************************************************)
	Event.no[1].Flag 										:= NOT Status_ReadyToEnable; Event.no[1].Class := TC2_SYSTEM.TCEVENTCLASS_HINT;
	Event.no[2].Flag 										:= Status_SyncError;
	Event.no[3].Flag 										:= Status_Error;
	Event.no[4].Flag 										:= Status_Warning; 				Event.no[4].Class := TC2_SYSTEM.TCEVENTCLASS_WARNING;
	Event.no[5].Flag 										:= Status_MotorStall AND FALSE;				Event.no[5].Class := TC2_SYSTEM.TCEVENTCLASS_STATEINFO;
	Event.no[6].Flag 										:= FALSE;
	Event.no[7].Flag 										:= ErrorSchutzschalter;
	Event.no[8].Flag 										:= ErrorEndlagePos; 	
	Event.no[9].Flag 										:= ErrorEndlageNeg;
	Event.no[10].Flag										:= FALSE; 					
(*	Event.no[11].Flag 										:= FALSE; 				
	Event.no[12].Flag 										:= FALSE;					
	Event.no[13].Flag 										:= FALSE; 			Event.no[9].Class := TC2_SYSTEM.TCEVENTCLASS_WARNING;
	Event.no[14].Flag 										:= FALSE; 			Event.no[10].Class := TC2_SYSTEM.TCEVENTCLASS_WARNING;
	Event.no[15].Flag 										:= FALSE;
	Event.no[16].Flag 										:= FALSE;
	Event.no[17].Flag 										:= FALSE;
	Event.no[18].Flag 										:= FALSE;
	Event.no[19].Flag 										:= FALSE;
	Event.no[20].Flag 										:= FALSE;
	Event.no[21].Flag 										:= FALSE;
	Event.no[22].Flag 										:= FALSE;
	Event.no[23].Flag 										:= FALSE;
	Event.no[24].Flag 										:= FALSE;
	Event.no[25].Flag 										:= FALSE;
*)
(* Check if msg activ and init some parameter ***********************)
	IF Event.no[1].Text2 <> Name OR Event.no[1].Text2 <> ''
	THEN
		(* Init Achsname *)
		FOR i := Event.MIN_EVENT TO Event.MAX_EVENT DO
		(*	Event.no[i].Text1								:= '';*)
			Event.no[i].Text2								:= SEL(LEN(name)>1,CONCAT('Axis id:',DWORD_TO_STRING(rAxis.NcToPlc.AxisId)),name);
		END_FOR
	END_IF

(* workl Event Ctrl *************************************************)
	Event(
		InAck 		:= InAck,
		Disable		:= rAxis.NcToPlc.AxisId = 0 OR NOT EnableEvent,
		SourceId	:= SOURCE_DRIVES_STEPPER + rAxis.NcToPlc.AxisId,
		HintActiv	=> ,
		MsgActiv	=> ,
		ErrActiv	=> ,
		AckRequired	=> ,
		StatusByte 	=> EventStatusByte);

(******************************************************************************)

METHOD PUBLIC Ack : bool
VAR_INPUT
END_VAR
Event.Ack();
END_METHOD

END_FUNCTION_BLOCK

// ---- POUs/PTP/02_Options/Parameter/AX_PARA_SET_ISTPOS.TcPOU
{attribute 'no_check'}
FUNCTION_BLOCK AX_PARA_SET_ISTPOS (* Datatyp - Set Istpos *)
VAR_INPUT
	Typ														: UDINT := 1; (* 0	NICHT DEFINIERT Wert wird nicht geschrieben
																			1	Absolutposition
																			2	Relativposition
																			5	Moduloposition *)
	Value													: LREAL;
END_VAR
VAR_OUTPUT
END_VAR
VAR
END_VAR

;

END_FUNCTION_BLOCK

// ---- POUs/PTP/02_Options/TouchProbe/Ax_TouchProbeCtrl.TcPOU
{attribute 'no_check'}
FUNCTION_BLOCK Ax_TouchProbeCtrl  (* Benötigte Lib: TcMC2.lib Version 2 - oder "Vom Uebersetzen ausschließen" aktivieren *)
VAR_OUTPUT CONSTANT
	FNC_RUN													:	INT := 0;
	FNC_ABORT												:	INT := 1;
END_VAR                     								
VAR_INPUT                   								
	Execute													:	BOOL := FALSE;
	Fnc														: 	INT (FNC_RUN..FNC_ABORT):= FNC_RUN;
	rAxis													: 	REFERENCE TO AXIS_REF := 0;
	TriggerInput											: 	TRIGGER_REF;
	WindowOnly												: 	BOOL := FALSE;(* Enables the monitoring window *)
	FirstPosition											: 	LREAL;	(* Beginning of the monitoring window *)
	LastPosition 											: 	LREAL;	(* Ending of the monitoring window *)
END_VAR
VAR_IN_OUT
END_VAR
VAR_OUTPUT
	Busy													:	BOOL;
	CmdAborted 												: 	BOOL;
	Done													: 	BOOL;	// will be TRUE, if axispositon is registered successfully
	Error													:	BOOL;
	ErrorId													:	UDINT;
	RecordedPosition										: 	LREAL;	// current axisposition on trigger-event
	RecordedData											:	MC_TouchProbeRecordedData;
END_VAR
VAR
(* cache **************************************************************************)
	MemFnc													:	INT := -1;
               								                           	
(* trigger *)               	
	rtExecute												:	R_TRIG;

(* MC-function-block instances ****************************************************)
	MC_TouchProbe											: 	MC_TouchProbe;
	MC_AbortTrigger											:	MC_AbortTrigger;

END_VAR

	(************************************************************************************)
	(*																					*)
	(*		B E C K H O F F   N E W   A U T O M A T I O N   T E C H N O L O G Y    		*)
	(*																					*)
	(*		Eiserstr.5	D-33415 Verl	Germany	phone:	+49-5246-0	www.Beckhoff.Com	*)
    (*																					*)
    (*		Bausteinbeschreibung	:	TouchProbe ctrl									*)
	(*		TwinCAT-Version			:	3.x or higher 									*)
	(*		Version					:	V3.0 / 03/13									*)
	(*		Lib						:	TcMC2.lib 										*)
 	(*		Autor					:	DSC												*)
	(*																					*)
	(************************************************************************************)

(* Execute ***************************************************************************************)
	rtExecute(CLK := Execute);
	IF rtExecute.Q
		AND MemFnc < 0
	THEN
		MemFnc 												:= SEL(Fnc = FNC_RUN, FNC_ABORT , FNC_RUN) ;
		Busy												:= TRUE;
		Done												:= FALSE;
		Error												:= FALSE;
		ErrorID												:= 0;
		CmdAborted											:= FALSE;
	END_IF

(* Call Method ***********************************************************************************)
	CASE MemFnc OF
	FNC_RUN:
		Run(Execute);

	FNC_ABORT:
		Abort(Execute);

	-1:
		IF NOT Execute
		THEN
			Busy											:= FALSE;
			Done											:= FALSE;
			Error											:= FALSE;
			ErrorID											:= 0;
			CmdAborted										:= FALSE;
		END_IF                              				
	ELSE                                    				
		Busy												:= FALSE;
		Done												:= FALSE;
		Error												:= Execute;
		ErrorID												:= 1803;
		CmdAborted											:= FALSE;
	END_CASE                                	

(*************************************************************************************************)

METHOD PUBLIC Abort : BOOL //Result = Busy
//required parameter
//rAxis
//TriggerInput
VAR_INPUT
	Execute													:	BOOL := FALSE;
END_VAR
	MemFnc	 												:= FNC_ABORT;
	THIS^.Execute											:= Execute;
IF NOT __ISVALIDREF(rAxis) 
THEN
	Busy													:= NOT Error;
	ErrorId													:= 16#4B30;
	Error													:= TRUE;
	Done													:= FALSE;
	CmdAborted												:= FALSE;
	MemFnc													:= SEL(Execute , -1 ,MemFnc); 
	RETURN;
END_IF

	MC_AbortTrigger(
		Execute		:= Execute,
		Axis		:= rAxis,
		TriggerInput:= TriggerInput,
		Done		=> done,
		Busy		=> Busy,
		Error		=> Error,
		ErrorID		=> ErrorID);

	CmdAborted		:= FALSE;

	IF NOT Execute AND NOT Busy
	THEN
		MemFnc												:= -1;
	END_IF                              					
	                                    	
	Abort 													:= Busy;
END_METHOD

METHOD PUBLIC Run : BOOL //Result = Busy
//required parameter
//rAxis
//TriggerInput
//WindowOnly
//FirstPosition
//LastPosition
VAR_INPUT
	Execute													: BOOL := FALSE;
END_VAR
	MemFnc 													:= FNC_RUN;
	THIS^.Execute											:= Execute;
	
IF NOT __ISVALIDREF(rAxis) 
THEN
	Busy													:= NOT Error;
	ErrorId													:= 16#4B30;
	Error													:= TRUE;
	Done													:= FALSE;
	CmdAborted												:= FALSE;
	MemFnc													:= SEL(Execute , -1 ,MemFnc); 
	RETURN;
END_IF

	MC_TouchProbe(
		Execute			:= Execute,
		WindowOnly		:= WindowOnly,
		FirstPosition	:= FirstPosition,
		LastPosition	:= LastPosition,
		Axis			:= rAxis,
		TriggerInput	:= TriggerInput,
		Done			=> Done,
		Busy			=> Busy,
		CommandAborted	=> CmdAborted,
		Error			=> Error,
		ErrorID			=> ErrorID,
		RecordedPosition=> RecordedPosition,
		RecordedData 	=> RecordedData);

	IF NOT Execute AND NOT Busy
	THEN
		MemFnc												:= -1;
	END_IF
END_METHOD

END_FUNCTION_BLOCK

// ---- POUs/PTP/03_Utilities/Ax_LoopingDistanceCtrl.TcPOU
FUNCTION_BLOCK Ax_LoopingDistanceCtrl (* Der Baustein ist nur für Eil/Schleichachsen gedacht !! *)
(* Schleifenweg:
	Bei Aktivierten Schleifenweg und z.B. einem Positiven Schleifenweg, wird das Ziel um den Schleifenweg ueberfahren und die Achse
	in Negative Richtung auf den Sollwert positioniert.
	Bei einer Positionerung in Negative Richtung wird das Ziel direkt angefahren. 
	Ist z.B die Achse im schon im Bremsbereich wird automatisch der Schleifenweg in aus der richtigen richtung aktiviert,
	damit die Achse nocheinmal die Zielpos. anfahren kann.
*)
VAR_OUTPUT CONSTANT
	FNC_OFF													:	INT := 0; (*	0 = Schleifenweg Aus *)
	FNC_AUTO												:	INT := 1; (*	1 = Schleifenweg Automatik - Der Schleifenweg wird
																						nur Aktiviert wenn die Achse innerhalb des Bremswegs ist.
																						Die Richtung wird aus SW-Endlagen und Versatz zum Sollwert ermittelt. *)
	FNC_POS_DIR												:	INT := 2; (* 2 = Schleifenweg Ein, ist der Schleifenweg 0 wird der Automatisch ermittelte Wert als Positiver Schleifenweg gesetzt *)
	FNC_NEG_DIR												:	INT := 3; (* 3 = Schleifenweg Ein, ist der Schleifenweg 0 wird der Automatisch ermittelte Wert als Neagtiver Schleifenweg gesetzt *)
END_VAR                             						
VAR_INPUT                           						
	Execute													:	BOOL := FALSE;	(* mit einem Positiven Signal wird der Baustein gestartet *)
	AxID													:	DWORD;				(* ID der Achse *)
	Mode													:	INT := FNC_AUTO;
	Istwert													:	LREAL;				(* Istwert der Achse *)
	Sollwert												:	LREAL;				(* Sollwert der Achse *)
	Schleifenweg											:	LREAL := 0;		(*	Sollwert Schleifenweg, Ist der Sollwert 0 wird er Automatisch aus
																							Bremsweg + (Schleichweg * 0.5) ermittelt (Min Schleifenweg) *)
	SWEndlagePos											: 	LREAL;
	SWEndlageNeg											: 	LREAL;
END_VAR                             						
VAR_OUTPUT                          						
	Busy													: 	BOOL;					(* Baustein in Bearbeitung *)
	Done													: 	BOOL;					(* Baustein hat Berabeitung beendet *)
	Error													: 	BOOL;					(* Im Baustein ist ein Fehler aufgetreten *)
	ErrorID													: 	UDINT;					(* Error ID der ADS Bausteine , Bei Error = True und ID <0 ist der Baustein nicht Richtig parametriert *)
END_VAR
VAR
(* ADS Read Write deklaration ***************************************************)
	MemErrorState											:	INT;
	ReadAds													: 	ADSREAD;
	WriteAds												: 	ADSWRITE;
	RT_Execute												: 	R_TRIG;

(* Zwischenspeicher *************************************************************)
	state													: 	INT := 0;
	iValue													: 	INT ;
	tmpSchleifenwegPos										: 	LREAL;
	tmpSchleifenwegNeg										: 	LREAL;
	tmpSchleifenweg											: 	LREAL;
	BremswegPos												: 	LREAL;
	BremswegNeg												: 	LREAL;
	SchleichwegPos											: 	LREAL;
	SchleichwegNeg											: 	LREAL;
END_VAR

(* Ax_LoopingDistanceCtrl																							*)
(* Schleifenweg automatisch anpassen und aktivieren - Eil/Schleichachse Ctrl V1.0									*)
(* Daniel Schlingmann																								*)
(********************************************************************************************************************)

(* Start Baustein *********************************************************************************)
RT_Execute(CLK := Execute);
CASE state OF
0:
	Busy 													:= FALSE;
	IF RT_Execute.Q 
	THEN
		Done 												:= FALSE;
		Busy 												:= TRUE;
		ReadAds	(Read := FALSE);
		WriteAds(Write := FALSE);

